LIN {X 0,Y 347.615,Z 494.435,A -85,B 0,C 180,E1 -13747.41,E2 -13747.41} C_VEL
LIN {X 0,Y 347.369,Z 499.212,A -85,B 0,C 180,E1 -13749.012,E2 -13749.012} C_VEL
LIN {X 0,Y 349.392,Z 514.132,A -85,B 0,C 180,E1 -13749.644,E2 -13749.644} C_VEL
LIN {X 0,Y 350.542,Z 527.666,A -85,B 0,C 180,E1 -13750.442,E2 -13750.442} C_VEL
LIN {X 0,Y 350.977,Z 539.209,A -85,B 0,C 180,E1 -13751.314,E2 -13751.314} C_VEL
LIN {X 0,Y 351.131,Z 550.524,A -85,B 0,C 180,E1 -13752.378,E2 -13752.378} C_VEL
LIN {X 0,Y 350.226,Z 559.587,A -85,B 0,C 180,E1 -13753.384,E2 -13753.384} C_VEL
LIN {X 0,Y 349.097,Z 570.237,A -85,B 0,C 180,E1 -13754.828,E2 -13754.828} C_VEL
LIN {X 0,Y 348.343,Z 577.267,A -85,B 0,C 180,E1 -13755.989,E2 -13755.989} C_VEL
LIN {X 0,Y 347.516,Z 586.102,A -85,B 0,C 180,E1 -13757.74,E2 -13757.74} C_VEL
LIN {X 0,Y 346.973,Z 593.197,A -85,B 0,C 180,E1 -13759.496,E2 -13759.496} C_VEL
LIN {X 0,Y 346.818,Z 598.935,A -85,B 0,C 180,E1 -13761.258,E2 -13761.258} C_VEL
LIN {X 0,Y 346.825,Z 603.831,A -85,B 0,C 180,E1 -13763.183,E2 -13763.183} C_VEL
LIN {X 0,Y 347.091,Z 607.836,A -85,B 0,C 180,E1 -13765.354,E2 -13765.354} C_VEL
LIN {X 0,Y 347.195,Z 609.309,A -85,B 0,C 180,E1 -13766.519,E2 -13766.519} C_VEL
LIN {X 0,Y 347.265,Z 610.359,A -85,B 0,C 180,E1 -13767.68,E2 -13767.68} C_VEL
LIN {X 0,Y 347.626,Z 611.268,A -85,B 0,C 180,E1 -13770,E2 -13770} C_VEL
LIN {X 0,Y 347.266,Z 610.353,A -85,B 0,C 180,E1 -13772.32,E2 -13772.32} C_VEL
LIN {X 0,Y 347.196,Z 609.302,A -85,B 0,C 180,E1 -13773.482,E2 -13773.482} C_VEL
LIN {X 0,Y 347.09,Z 607.824,A -85,B 0,C 180,E1 -13774.646,E2 -13774.646} C_VEL
LIN {X 0,Y 346.813,Z 603.843,A -85,B 0,C 180,E1 -13776.8,E2 -13776.8} C_VEL
LIN {X 0,Y 346.818,Z 598.902,A -85,B 0,C 180,E1 -13778.742,E2 -13778.742} C_VEL
LIN {X 0,Y 346.977,Z 593.158,A -85,B 0,C 180,E1 -13780.504,E2 -13780.504} C_VEL
LIN {X 0,Y 347.512,Z 586.051,A -85,B 0,C 180,E1 -13782.26,E2 -13782.26} C_VEL
LIN {X 0,Y 348.302,Z 577.193,A -85,B 0,C 180,E1 -13784.013,E2 -13784.013} C_VEL
LIN {X 0,Y 349.339,Z 568.176,A -85,B 0,C 180,E1 -13785.46,E2 -13785.46} C_VEL
LIN {X 0,Y 350.409,Z 558.302,A -85,B 0,C 180,E1 -13786.757,E2 -13786.757} C_VEL
LIN {X 0,Y 351.091,Z 550.396,A -85,B 0,C 180,E1 -13787.624,E2 -13787.624} C_VEL
LIN {X 0,Y 350.986,Z 539.051,A -85,B 0,C 180,E1 -13788.686,E2 -13788.686} C_VEL
LIN {X 0,Y 350.444,Z 525.95,A -85,B 0,C 180,E1 -13789.661,E2 -13789.661} C_VEL
LIN {X 0,Y 349.17,Z 512.232,A -85,B 0,C 180,E1 -13790.432,E2 -13790.432} C_VEL
LIN {X 0,Y 347.349,Z 499.21,A -85,B 0,C 180,E1 -13790.97,E2 -13790.97} C_VEL
LIN {X 0,Y 348.076,Z 488.085,A -85,B 0,C 180,E1 -13794.688,E2 -13794.688} C_VEL
LIN {X 0,Y 349.057,Z 475.439,A -85,B 0,C 180,E1 -13798.896,E2 -13798.896} C_VEL
LIN {X 0,Y 350.254,Z 463.775,A -85,B 0,C 180,E1 -13802.804,E2 -13802.804} C_VEL
LIN {X 0,Y 351.609,Z 451.807,A -85,B 0,C 180,E1 -13806.915,E2 -13806.915} C_VEL
LIN {X 0,Y 351.655,Z 448.004,A -85,B 0,C 180,E1 -13808.284,E2 -13808.284} C_VEL
LIN {X 0,Y 350.132,Z 439.763,A -85,B 0,C 180,E1 -13811.483,E2 -13811.483} C_VEL
LIN {X 0,Y 348.357,Z 431.103,A -85,B 0,C 180,E1 -13815.08,E2 -13815.08} C_VEL
LIN {X 0,Y 347.734,Z 428.173,A -85,B 0,C 180,E1 -13816.394,E2 -13816.394} C_VEL
LIN {X 0,Y 347.735,Z 428.172,A -85,B 0,C 180,E1 -13819.703,E2 -13819.703} C_VEL
LIN {X 0,Y 347.765,Z 428.164,A -85,B 0,C 180,E1 -13822.68,E2 -13822.68} C_VEL
LIN {X 0,Y 347.751,Z 428.17,A -85,B 0,C 180,E1 -13825.956,E2 -13825.956} C_VEL
LIN {X 0,Y 347.752,Z 428.167,A -85,B 0,C 180,E1 -13829.652,E2 -13829.652} C_VEL
LIN {X 0,Y 347.833,Z 428.157,A -85,B 0,C 180,E1 -13833.608,E2 -13833.608} C_VEL
LIN {X 0,Y 347.787,Z 428.164,A -85,B 0,C 180,E1 -13836.162,E2 -13836.162} C_VEL
LIN {X 0,Y 347.815,Z 428.162,A -85,B 0,C 180,E1 -13839.909,E2 -13839.909} C_VEL
LIN {X 0,Y 347.87,Z 428.151,A -85,B 0,C 180,E1 -13842.359,E2 -13842.359} C_VEL
LIN {X 0,Y 347.901,Z 428.15,A -85,B 0,C 180,E1 -13845.971,E2 -13845.971} C_VEL
LIN {X 0,Y 347.933,Z 428.146,A -85,B 0,C 180,E1 -13849.526,E2 -13849.526} C_VEL
LIN {X 0,Y 348.083,Z 428.124,A -85,B 0,C 180,E1 -13853.042,E2 -13853.042} C_VEL
LIN {X 0,Y 348.212,Z 428.113,A -85,B 0,C 180,E1 -13857.687,E2 -13857.687} C_VEL
LIN {X 0,Y 348.371,Z 428.089,A -85,B 0,C 180,E1 -13860,E2 -13860} C_VEL
LIN {X 0,Y 348.21,Z 428.108,A -85,B 0,C 180,E1 -13862.314,E2 -13862.314} C_VEL
LIN {X 0,Y 348.082,Z 428.124,A -85,B 0,C 180,E1 -13866.958,E2 -13866.958} C_VEL
LIN {X 0,Y 347.934,Z 428.141,A -85,B 0,C 180,E1 -13870.474,E2 -13870.474} C_VEL
LIN {X 0,Y 347.901,Z 428.143,A -85,B 0,C 180,E1 -13874.15,E2 -13874.15} C_VEL
LIN {X 0,Y 347.894,Z 428.145,A -85,B 0,C 180,E1 -13878.29,E2 -13878.29} C_VEL
LIN {X 0,Y 347.793,Z 428.162,A -85,B 0,C 180,E1 -13881.636,E2 -13881.636} C_VEL
LIN {X 0,Y 347.816,Z 428.159,A -85,B 0,C 180,E1 -13885.108,E2 -13885.108} C_VEL
LIN {X 0,Y 347.811,Z 428.156,A -85,B 0,C 180,E1 -13887.694,E2 -13887.694} C_VEL
LIN {X 0,Y 347.752,Z 428.163,A -85,B 0,C 180,E1 -13890.348,E2 -13890.348} C_VEL
LIN {X 0,Y 347.751,Z 428.164,A -85,B 0,C 180,E1 -13894.044,E2 -13894.044} C_VEL
LIN {X 0,Y 347.764,Z 428.167,A -85,B 0,C 180,E1 -13897.321,E2 -13897.321} C_VEL
LIN {X 0,Y 347.735,Z 428.166,A -85,B 0,C 180,E1 -13900.297,E2 -13900.297} C_VEL
LIN {X 0,Y 347.732,Z 428.169,A -85,B 0,C 180,E1 -13903.407,E2 -13903.407} C_VEL
LIN {X 0,Y 347.788,Z 428.162,A -85,B 0,C 180,E1 -13906.676,E2 -13906.676} C_VEL
LIN {X 0,Y 347.789,Z 428.159,A -85,B 0,C 180,E1 -13910.165,E2 -13910.165} C_VEL
LIN {X 0,Y 347.793,Z 428.159,A -85,B 0,C 180,E1 -13914.125,E2 -13914.125} C_VEL
LIN {X 0,Y 347.741,Z 428.165,A -85,B 0,C 180,E1 -13918.086,E2 -13918.086} C_VEL
LIN {X 0,Y 347.782,Z 428.166,A -85,B 0,C 180,E1 -13920.988,E2 -13920.988} C_VEL
LIN {X 0,Y 347.834,Z 428.155,A -85,B 0,C 180,E1 -13923.608,E2 -13923.608} C_VEL
LIN {X 0,Y 347.792,Z 428.16,A -85,B 0,C 180,E1 -13926.162,E2 -13926.162} C_VEL
LIN {X 0,Y 347.82,Z 428.157,A -85,B 0,C 180,E1 -13929.91,E2 -13929.91} C_VEL
LIN {X 0,Y 347.858,Z 428.349,A -85,B 0,C 180,E1 -13930.016,E2 -13930.016} C_VEL
LIN {X 0,Y 351.858,Z 440.054,A -85,B 0,C 180,E1 -13931.095,E2 -13931.095} C_VEL
LIN {X 0,Y 354.541,Z 449.162,A -85,B 0,C 180,E1 -13932.082,E2 -13932.082} C_VEL
LIN {X 0,Y 355.019,Z 451.116,A -85,B 0,C 180,E1 -13932.305,E2 -13932.305} C_VEL
LIN {X 0,Y 354.008,Z 461.436,A -85,B 0,C 180,E1 -13933.418,E2 -13933.418} C_VEL
LIN {X 0,Y 353.05,Z 471.021,A -85,B 0,C 180,E1 -13934.706,E2 -13934.706} C_VEL
LIN {X 0,Y 352.106,Z 479.723,A -85,B 0,C 180,E1 -13936.142,E2 -13936.142} C_VEL
LIN {X 0,Y 350.939,Z 488.223,A -85,B 0,C 180,E1 -13937.861,E2 -13937.861} C_VEL
LIN {X 0,Y 349.95,Z 495.551,A -85,B 0,C 180,E1 -13939.758,E2 -13939.758} C_VEL
LIN {X 0,Y 349.449,Z 500.347,A -85,B 0,C 180,E1 -13941.324,E2 -13941.324} C_VEL
LIN {X 0,Y 348.745,Z 504.594,A -85,B 0,C 180,E1 -13943.055,E2 -13943.055} C_VEL
LIN {X 0,Y 348.436,Z 506.829,A -85,B 0,C 180,E1 -13944.212,E2 -13944.212} C_VEL
LIN {X 0,Y 348.162,Z 508.651,A -85,B 0,C 180,E1 -13945.369,E2 -13945.369} C_VEL
LIN {X 0,Y 347.931,Z 510.025,A -85,B 0,C 180,E1 -13946.526,E2 -13946.526} C_VEL
LIN {X 0,Y 347.95,Z 511.562,A -85,B 0,C 180,E1 -13948.843,E2 -13948.843} C_VEL
LIN {X 0,Y 347.949,Z 511.785,A -85,B 0,C 180,E1 -13950,E2 -13950} C_VEL
LIN {X 0,Y 347.949,Z 511.603,A -85,B 0,C 180,E1 -13951.157,E2 -13951.157} C_VEL
LIN {X 0,Y 347.923,Z 510.12,A -85,B 0,C 180,E1 -13953.474,E2 -13953.474} C_VEL
LIN {X 0,Y 348.151,Z 508.789,A -85,B 0,C 180,E1 -13954.631,E2 -13954.631} C_VEL
LIN {X 0,Y 348.63,Z 505.972,A -85,B 0,C 180,E1 -13956.366,E2 -13956.366} C_VEL
LIN {X 0,Y 349.241,Z 502.154,A -85,B 0,C 180,E1 -13958.098,E2 -13958.098} C_VEL
LIN {X 0,Y 349.841,Z 496.248,A -85,B 0,C 180,E1 -13960.143,E2 -13960.143} C_VEL
LIN {X 0,Y 350.782,Z 489.852,A -85,B 0,C 180,E1 -13961.851,E2 -13961.851} C_VEL
LIN {X 0,Y 351.886,Z 481.818,A -85,B 0,C 180,E1 -13963.572,E2 -13963.572} C_VEL
LIN {X 0,Y 352.754,Z 473.601,A -85,B 0,C 180,E1 -13965.011,E2 -13965.011} C_VEL
LIN {X 0,Y 353.83,Z 463.41,A -85,B 0,C 180,E1 -13966.442,E2 -13966.442} C_VEL
LIN {X 0,Y 354.776,Z 453.903,A -85,B 0,C 180,E1 -13967.519,E2 -13967.519} C_VEL
LIN {X 0,Y 354.989,Z 450.779,A -85,B 0,C 180,E1 -13967.836,E2 -13967.836} C_VEL
LIN {X 0,Y 351.781,Z 439.815,A -85,B 0,C 180,E1 -13969.035,E2 -13969.035} C_VEL
LIN {X 0,Y 347.808,Z 428.164,A -85,B 0,C 180,E1 -13970.129,E2 -13970.129} C_VEL
LIN {X 0,Y 347.791,Z 428.161,A -85,B 0,C 180,E1 -13973.838,E2 -13973.838} C_VEL
LIN {X 0,Y 347.852,Z 428.157,A -85,B 0,C 180,E1 -13977.255,E2 -13977.255} C_VEL
LIN {X 0,Y 347.751,Z 428.164,A -85,B 0,C 180,E1 -13980.348,E2 -13980.348} C_VEL
LIN {X 0,Y 347.75,Z 428.164,A -85,B 0,C 180,E1 -13984.044,E2 -13984.044} C_VEL
LIN {X 0,Y 347.769,Z 428.166,A -85,B 0,C 180,E1 -13987.32,E2 -13987.32} C_VEL
LIN {X 0,Y 347.796,Z 428.159,A -85,B 0,C 180,E1 -13990.288,E2 -13990.288} C_VEL
LIN {X 0,Y 347.788,Z 428.162,A -85,B 0,C 180,E1 -13993.398,E2 -13993.398} C_VEL
LIN {X 0,Y 347.732,Z 428.17,A -85,B 0,C 180,E1 -13996.685,E2 -13996.685} C_VEL
LIN {X 0,Y 347.738,Z 428.166,A -85,B 0,C 180,E1 -13999.9,E2 -13999.9} C_VEL
LIN {X 0,Y 347.096,Z 428.251,A -85,B 0,C 180,E1 -14000.867,E2 -14000.867} C_VEL
LIN {X 0,Y 344.256,Z 428.605,A -85,B 0,C 180,E1 -14002.441,E2 -14002.441} C_VEL
LIN {X 0,Y 341.835,Z 428.908,A -85,B 0,C 180,E1 -14003.715,E2 -14003.715} C_VEL
LIN {X 0,Y 340.796,Z 429.035,A -85,B 0,C 180,E1 -14004.701,E2 -14004.701} C_VEL
LIN {X 0,Y 340.712,Z 429.043,A -85,B 0,C 180,E1 -14005.034,E2 -14005.034} C_VEL
LIN {X 0,Y 340.7,Z 429.048,A -85,B 0,C 180,E1 -14008.955,E2 -14008.955} C_VEL
LIN {X 0,Y 340.805,Z 429.033,A -85,B 0,C 180,E1 -14013.02,E2 -14013.02} C_VEL
LIN {X 0,Y 340.758,Z 429.035,A -85,B 0,C 180,E1 -14015.638,E2 -14015.638} C_VEL
LIN {X 0,Y 340.755,Z 429.036,A -85,B 0,C 180,E1 -14019.475,E2 -14019.475} C_VEL
LIN {X 0,Y 340.86,Z 429.023,A -85,B 0,C 180,E1 -14021.984,E2 -14021.984} C_VEL
LIN {X 0,Y 340.871,Z 429.021,A -85,B 0,C 180,E1 -14025.705,E2 -14025.705} C_VEL
LIN {X 0,Y 340.875,Z 429.021,A -85,B 0,C 180,E1 -14029.306,E2 -14029.306} C_VEL
LIN {X 0,Y 341.051,Z 429,A -85,B 0,C 180,E1 -14032.898,E2 -14032.898} C_VEL
LIN {X 0,Y 341.173,Z 428.984,A -85,B 0,C 180,E1 -14037.639,E2 -14037.639} C_VEL
LIN {X 0,Y 341.319,Z 428.968,A -85,B 0,C 180,E1 -14040,E2 -14040} C_VEL
LIN {X 0,Y 341.173,Z 428.988,A -85,B 0,C 180,E1 -14042.361,E2 -14042.361} C_VEL
LIN {X 0,Y 341.049,Z 428.999,A -85,B 0,C 180,E1 -14047.102,E2 -14047.102} C_VEL
LIN {X 0,Y 340.875,Z 429.023,A -85,B 0,C 180,E1 -14050.694,E2 -14050.694} C_VEL
LIN {X 0,Y 340.865,Z 429.027,A -85,B 0,C 180,E1 -14054.325,E2 -14054.325} C_VEL
LIN {X 0,Y 340.84,Z 429.029,A -85,B 0,C 180,E1 -14058.467,E2 -14058.467} C_VEL
LIN {X 0,Y 340.719,Z 429.044,A -85,B 0,C 180,E1 -14061.842,E2 -14061.842} C_VEL
LIN {X 0,Y 340.773,Z 429.036,A -85,B 0,C 180,E1 -14065.664,E2 -14065.664} C_VEL
LIN {X 0,Y 340.731,Z 429.042,A -85,B 0,C 180,E1 -14068.321,E2 -14068.321} C_VEL
LIN {X 0,Y 340.699,Z 429.043,A -85,B 0,C 180,E1 -14071.045,E2 -14071.045} C_VEL
LIN {X 0,Y 340.72,Z 429.042,A -85,B 0,C 180,E1 -14075.279,E2 -14075.279} C_VEL
LIN {X 0,Y 340.712,Z 429.044,A -85,B 0,C 180,E1 -14078.386,E2 -14078.386} C_VEL
LIN {X 0,Y 340.701,Z 429.05,A -85,B 0,C 180,E1 -14082.046,E2 -14082.046} C_VEL
LIN {X 0,Y 340.693,Z 429.067,A -85,B 0,C 180,E1 -14083.145,E2 -14083.145} C_VEL
LIN {X 0,Y 342.387,Z 437.143,A -85,B 0,C 180,E1 -14086.699,E2 -14086.699} C_VEL
LIN {X 0,Y 343.982,Z 445.1,A -85,B 0,C 180,E1 -14089.972,E2 -14089.972} C_VEL
LIN {X 0,Y 344.84,Z 451.146,A -85,B 0,C 180,E1 -14092.308,E2 -14092.308} C_VEL
LIN {X 0,Y 343.637,Z 460.942,A -85,B 0,C 180,E1 -14095.776,E2 -14095.776} C_VEL
LIN {X 0,Y 342.775,Z 468.732,A -85,B 0,C 180,E1 -14098.478,E2 -14098.478} C_VEL
LIN {X 0,Y 341.626,Z 480.835,A -85,B 0,C 180,E1 -14102.627,E2 -14102.627} C_VEL
LIN {X 0,Y 340.803,Z 491.561,A -85,B 0,C 180,E1 -14106.289,E2 -14106.289} C_VEL
LIN {X 0,Y 340.351,Z 498.191,A -85,B 0,C 180,E1 -14108.568,E2 -14108.568} C_VEL
LIN {X 0,Y 342.379,Z 512.492,A -85,B 0,C 180,E1 -14109.184,E2 -14109.184} C_VEL
LIN {X 0,Y 343.496,Z 525.586,A -85,B 0,C 180,E1 -14109.955,E2 -14109.955} C_VEL
LIN {X 0,Y 344.073,Z 538.171,A -85,B 0,C 180,E1 -14110.924,E2 -14110.924} C_VEL
LIN {X 0,Y 344.161,Z 550.943,A -85,B 0,C 180,E1 -14112.163,E2 -14112.163} C_VEL
LIN {X 0,Y 343.238,Z 559.759,A -85,B 0,C 180,E1 -14113.189,E2 -14113.189} C_VEL
LIN {X 0,Y 342.06,Z 570.288,A -85,B 0,C 180,E1 -14114.686,E2 -14114.686} C_VEL
LIN {X 0,Y 341.269,Z 577.873,A -85,B 0,C 180,E1 -14115.997,E2 -14115.997} C_VEL
LIN {X 0,Y 340.406,Z 586.348,A -85,B 0,C 180,E1 -14117.783,E2 -14117.783} C_VEL
LIN {X 0,Y 339.886,Z 593.222,A -85,B 0,C 180,E1 -14119.576,E2 -14119.576} C_VEL
LIN {X 0,Y 339.731,Z 599.572,A -85,B 0,C 180,E1 -14121.674,E2 -14121.674} C_VEL
LIN {X 0,Y 339.756,Z 603.095,A -85,B 0,C 180,E1 -14123.17,E2 -14123.17} C_VEL
LIN {X 0,Y 340.028,Z 606.823,A -85,B 0,C 180,E1 -14125.258,E2 -14125.258} C_VEL
LIN {X 0,Y 340.147,Z 608.299,A -85,B 0,C 180,E1 -14126.446,E2 -14126.446} C_VEL
LIN {X 0,Y 340.221,Z 609.351,A -85,B 0,C 180,E1 -14127.632,E2 -14127.632} C_VEL
LIN {X 0,Y 340.597,Z 610.263,A -85,B 0,C 180,E1 -14130,E2 -14130} C_VEL
LIN {X 0,Y 340.222,Z 609.345,A -85,B 0,C 180,E1 -14132.368,E2 -14132.368} C_VEL
LIN {X 0,Y 340.147,Z 608.291,A -85,B 0,C 180,E1 -14133.554,E2 -14133.554} C_VEL
LIN {X 0,Y 340.027,Z 606.81,A -85,B 0,C 180,E1 -14134.743,E2 -14134.743} C_VEL
LIN {X 0,Y 339.75,Z 603.089,A -85,B 0,C 180,E1 -14136.821,E2 -14136.821} C_VEL
LIN {X 0,Y 339.742,Z 597.877,A -85,B 0,C 180,E1 -14138.925,E2 -14138.925} C_VEL
LIN {X 0,Y 339.937,Z 592.133,A -85,B 0,C 180,E1 -14140.724,E2 -14140.724} C_VEL
LIN {X 0,Y 340.505,Z 585.023,A -85,B 0,C 180,E1 -14142.517,E2 -14142.517} C_VEL
LIN {X 0,Y 341.232,Z 577.802,A -85,B 0,C 180,E1 -14144.005,E2 -14144.005} C_VEL
LIN {X 0,Y 342.036,Z 570.341,A -85,B 0,C 180,E1 -14145.293,E2 -14145.293} C_VEL
LIN {X 0,Y 343.041,Z 560.804,A -85,B 0,C 180,E1 -14146.668,E2 -14146.668} C_VEL
LIN {X 0,Y 344.134,Z 550.811,A -85,B 0,C 180,E1 -14147.839,E2 -14147.839} C_VEL
LIN {X 0,Y 344.045,Z 537.997,A -85,B 0,C 180,E1 -14149.077,E2 -14149.077} C_VEL
LIN {X 0,Y 343.509,Z 525.338,A -85,B 0,C 180,E1 -14150.045,E2 -14150.045} C_VEL
LIN {X 0,Y 342.262,Z 511.646,A -85,B 0,C 180,E1 -14150.843,E2 -14150.843} C_VEL
LIN {X 0,Y 340.324,Z 498.16,A -85,B 0,C 180,E1 -14151.422,E2 -14151.422} C_VEL
LIN {X 0,Y 341.221,Z 485.908,A -85,B 0,C 180,E1 -14155.628,E2 -14155.628} C_VEL
LIN {X 0,Y 342.144,Z 474.463,A -85,B 0,C 180,E1 -14159.537,E2 -14159.537} C_VEL
LIN {X 0,Y 343.266,Z 464.612,A -85,B 0,C 180,E1 -14162.92,E2 -14162.92} C_VEL
LIN {X 0,Y 344.722,Z 452.086,A -85,B 0,C 180,E1 -14167.334,E2 -14167.334} C_VEL
LIN {X 0,Y 344.678,Z 449.176,A -85,B 0,C 180,E1 -14168.408,E2 -14168.408} C_VEL
LIN {X 0,Y 343.159,Z 440.988,A -85,B 0,C 180,E1 -14171.664,E2 -14171.664} C_VEL
LIN {X 0,Y 341.562,Z 433.244,A -85,B 0,C 180,E1 -14174.955,E2 -14174.955} C_VEL
LIN {X 0,Y 340.674,Z 429.052,A -85,B 0,C 180,E1 -14176.854,E2 -14176.854} C_VEL
LIN {X 0,Y 340.702,Z 429.049,A -85,B 0,C 180,E1 -14180.248,E2 -14180.248} C_VEL
LIN {X 0,Y 340.713,Z 429.043,A -85,B 0,C 180,E1 -14183.559,E2 -14183.559} C_VEL
LIN {X 0,Y 340.697,Z 429.048,A -85,B 0,C 180,E1 -14186.154,E2 -14186.154} C_VEL
LIN {X 0,Y 340.744,Z 429.041,A -85,B 0,C 180,E1 -14190.329,E2 -14190.329} C_VEL
LIN {X 0,Y 340.806,Z 429.03,A -85,B 0,C 180,E1 -14193.02,E2 -14193.02} C_VEL
LIN {X 0,Y 340.757,Z 429.039,A -85,B 0,C 180,E1 -14195.638,E2 -14195.638} C_VEL
LIN {X 0,Y 340.74,Z 429.04,A -85,B 0,C 180,E1 -14199.474,E2 -14199.474} C_VEL
LIN {X 0,Y 340.861,Z 429.028,A -85,B 0,C 180,E1 -14201.984,E2 -14201.984} C_VEL
LIN {X 0,Y 340.872,Z 429.027,A -85,B 0,C 180,E1 -14205.705,E2 -14205.705} C_VEL
LIN {X 0,Y 340.876,Z 429.023,A -85,B 0,C 180,E1 -14209.306,E2 -14209.306} C_VEL
LIN {X 0,Y 341.05,Z 429,A -85,B 0,C 180,E1 -14212.898,E2 -14212.898} C_VEL
LIN {X 0,Y 341.174,Z 428.989,A -85,B 0,C 180,E1 -14217.639,E2 -14217.639} C_VEL
LIN {X 0,Y 341.32,Z 428.968,A -85,B 0,C 180,E1 -14220,E2 -14220} C_VEL
LIN {X 0,Y 341.172,Z 428.984,A -85,B 0,C 180,E1 -14222.361,E2 -14222.361} C_VEL
LIN {X 0,Y 341.05,Z 429.001,A -85,B 0,C 180,E1 -14227.102,E2 -14227.102} C_VEL
LIN {X 0,Y 340.877,Z 429.021,A -85,B 0,C 180,E1 -14230.694,E2 -14230.694} C_VEL
LIN {X 0,Y 340.866,Z 429.018,A -85,B 0,C 180,E1 -14234.325,E2 -14234.325} C_VEL
LIN {X 0,Y 340.84,Z 429.023,A -85,B 0,C 180,E1 -14238.466,E2 -14238.466} C_VEL
LIN {X 0,Y 340.757,Z 429.037,A -85,B 0,C 180,E1 -14241.857,E2 -14241.857} C_VEL
LIN {X 0,Y 340.776,Z 429.033,A -85,B 0,C 180,E1 -14245.664,E2 -14245.664} C_VEL
LIN {X 0,Y 340.731,Z 429.034,A -85,B 0,C 180,E1 -14248.321,E2 -14248.321} C_VEL
LIN {X 0,Y 340.701,Z 429.045,A -85,B 0,C 180,E1 -14251.045,E2 -14251.045} C_VEL
LIN {X 0,Y 340.721,Z 429.045,A -85,B 0,C 180,E1 -14255.279,E2 -14255.279} C_VEL
LIN {X 0,Y 340.712,Z 429.042,A -85,B 0,C 180,E1 -14258.386,E2 -14258.386} C_VEL
LIN {X 0,Y 340.702,Z 429.042,A -85,B 0,C 180,E1 -14262.046,E2 -14262.046} C_VEL
LIN {X 0,Y 340.724,Z 429.042,A -85,B 0,C 180,E1 -14265.468,E2 -14265.468} C_VEL
LIN {X 0,Y 340.728,Z 429.042,A -85,B 0,C 180,E1 -14268.696,E2 -14268.696} C_VEL
LIN {X 0,Y 340.744,Z 429.037,A -85,B 0,C 180,E1 -14271.774,E2 -14271.774} C_VEL
LIN {X 0,Y 340.726,Z 429.039,A -85,B 0,C 180,E1 -14275.595,E2 -14275.595} C_VEL
LIN {X 0,Y 340.7,Z 429.048,A -85,B 0,C 180,E1 -14278.955,E2 -14278.955} C_VEL
LIN {X 0,Y 340.806,Z 429.035,A -85,B 0,C 180,E1 -14283.02,E2 -14283.02} C_VEL
LIN {X 0,Y 340.759,Z 429.036,A -85,B 0,C 180,E1 -14285.638,E2 -14285.638} C_VEL
LIN {X 0,Y 340.763,Z 429.036,A -85,B 0,C 180,E1 -14289.543,E2 -14289.543} C_VEL
LIN {X 0,Y 344.712,Z 440.423,A -85,B 0,C 180,E1 -14290.631,E2 -14290.631} C_VEL
LIN {X 0,Y 347.762,Z 450.74,A -85,B 0,C 180,E1 -14291.776,E2 -14291.776} C_VEL
LIN {X 0,Y 348.214,Z 452.481,A -85,B 0,C 180,E1 -14291.983,E2 -14291.983} C_VEL
LIN {X 0,Y 347.178,Z 463.595,A -85,B 0,C 180,E1 -14293.234,E2 -14293.234} C_VEL
LIN {X 0,Y 346.063,Z 473.943,A -85,B 0,C 180,E1 -14294.692,E2 -14294.692} C_VEL
LIN {X 0,Y 345.095,Z 482.305,A -85,B 0,C 180,E1 -14296.155,E2 -14296.155} C_VEL
LIN {X 0,Y 343.912,Z 490.435,A -85,B 0,C 180,E1 -14297.909,E2 -14297.909} C_VEL
LIN {X 0,Y 343.036,Z 496.558,A -85,B 0,C 180,E1 -14299.55,E2 -14299.55} C_VEL
LIN {X 0,Y 342.504,Z 501.354,A -85,B 0,C 180,E1 -14301.147,E2 -14301.147} C_VEL
LIN {X 0,Y 341.772,Z 505.6,A -85,B 0,C 180,E1 -14302.913,E2 -14302.913} C_VEL
LIN {X 0,Y 341.445,Z 507.835,A -85,B 0,C 180,E1 -14304.093,E2 -14304.093} C_VEL
LIN {X 0,Y 341.157,Z 509.657,A -85,B 0,C 180,E1 -14305.273,E2 -14305.273} C_VEL
LIN {X 0,Y 340.916,Z 511.031,A -85,B 0,C 180,E1 -14306.454,E2 -14306.454} C_VEL
LIN {X 0,Y 340.931,Z 512.566,A -85,B 0,C 180,E1 -14308.819,E2 -14308.819} C_VEL
LIN {X 0,Y 340.928,Z 512.79,A -85,B 0,C 180,E1 -14310,E2 -14310} C_VEL
LIN {X 0,Y 340.931,Z 512.607,A -85,B 0,C 180,E1 -14311.181,E2 -14311.181} C_VEL
LIN {X 0,Y 340.909,Z 511.125,A -85,B 0,C 180,E1 -14313.546,E2 -14313.546} C_VEL
LIN {X 0,Y 341.146,Z 509.793,A -85,B 0,C 180,E1 -14314.727,E2 -14314.727} C_VEL
LIN {X 0,Y 341.648,Z 506.976,A -85,B 0,C 180,E1 -14316.496,E2 -14316.496} C_VEL
LIN {X 0,Y 342.284,Z 503.158,A -85,B 0,C 180,E1 -14318.264,E2 -14318.264} C_VEL
LIN {X 0,Y 342.924,Z 497.255,A -85,B 0,C 180,E1 -14320.349,E2 -14320.349} C_VEL
LIN {X 0,Y 343.907,Z 490.855,A -85,B 0,C 180,E1 -14322.091,E2 -14322.091} C_VEL
LIN {X 0,Y 345.058,Z 482.82,A -85,B 0,C 180,E1 -14323.846,E2 -14323.846} C_VEL
LIN {X 0,Y 345.971,Z 474.603,A -85,B 0,C 180,E1 -14325.312,E2 -14325.312} C_VEL
LIN {X 0,Y 347.095,Z 464.411,A -85,B 0,C 180,E1 -14326.77,E2 -14326.77} C_VEL
LIN {X 0,Y 348.141,Z 454.319,A -85,B 0,C 180,E1 -14327.927,E2 -14327.927} C_VEL
LIN {X 0,Y 348.212,Z 452.186,A -85,B 0,C 180,E1 -14328.155,E2 -14328.155} C_VEL
LIN {X 0,Y 344.956,Z 441.235,A -85,B 0,C 180,E1 -14329.396,E2 -14329.396} C_VEL
LIN {X 0,Y 340.788,Z 429.038,A -85,B 0,C 180,E1 -14330.563,E2 -14330.563} C_VEL
LIN {X 0,Y 340.769,Z 429.037,A -85,B 0,C 180,E1 -14334.844,E2 -14334.844} C_VEL
LIN {X 0,Y 340.778,Z 429.035,A -85,B 0,C 180,E1 -14337.525,E2 -14337.525} C_VEL
LIN {X 0,Y 340.7,Z 429.047,A -85,B 0,C 180,E1 -14341.044,E2 -14341.044} C_VEL
LIN {X 0,Y 340.721,Z 429.045,A -85,B 0,C 180,E1 -14345.279,E2 -14345.279} C_VEL
LIN {X 0,Y 340.727,Z 429.04,A -85,B 0,C 180,E1 -14348.389,E2 -14348.389} C_VEL
LIN {X 0,Y 340.728,Z 429.043,A -85,B 0,C 180,E1 -14351.303,E2 -14351.303} C_VEL
LIN {X 0,Y 340.724,Z 429.041,A -85,B 0,C 180,E1 -14354.532,E2 -14354.532} C_VEL
LIN {X 0,Y 340.688,Z 429.047,A -85,B 0,C 180,E1 -14358.691,E2 -14358.691} C_VEL
LIN {X 0,Y 340.735,Z 429.039,A -85,B 0,C 180,E1 -14361.773,E2 -14361.773} C_VEL
LIN {X 0,Y 340.712,Z 429.043,A -85,B 0,C 180,E1 -14365.034,E2 -14365.034} C_VEL
LIN {X 0,Y 340.049,Z 429.125,A -85,B 0,C 180,E1 -14366.021,E2 -14366.021} C_VEL
LIN {X 0,Y 337.206,Z 429.477,A -85,B 0,C 180,E1 -14367.626,E2 -14367.626} C_VEL
LIN {X 0,Y 334.794,Z 429.784,A -85,B 0,C 180,E1 -14368.925,E2 -14368.925} C_VEL
LIN {X 0,Y 333.758,Z 429.908,A -85,B 0,C 180,E1 -14369.931,E2 -14369.931} C_VEL
LIN {X 0,Y 333.673,Z 429.917,A -85,B 0,C 180,E1 -14370.271,E2 -14370.271} C_VEL
LIN {X 0,Y 333.737,Z 429.91,A -85,B 0,C 180,E1 -14373.754,E2 -14373.754} C_VEL
LIN {X 0,Y 333.721,Z 429.911,A -85,B 0,C 180,E1 -14377.914,E2 -14377.914} C_VEL
LIN {X 0,Y 333.796,Z 429.902,A -85,B 0,C 180,E1 -14381.589,E2 -14381.589} C_VEL
LIN {X 0,Y 333.81,Z 429.901,A -85,B 0,C 180,E1 -14385.576,E2 -14385.576} C_VEL
LIN {X 0,Y 333.838,Z 429.898,A -85,B 0,C 180,E1 -14389.078,E2 -14389.078} C_VEL
LIN {X 0,Y 333.997,Z 429.88,A -85,B 0,C 180,E1 -14392.747,E2 -14392.747} C_VEL
LIN {X 0,Y 333.811,Z 429.899,A -85,B 0,C 180,E1 -14395.169,E2 -14395.169} C_VEL
LIN {X 0,Y 334.11,Z 429.864,A -85,B 0,C 180,E1 -14397.589,E2 -14397.589} C_VEL
LIN {X 0,Y 334.269,Z 429.846,A -85,B 0,C 180,E1 -14400,E2 -14400} C_VEL
LIN {X 0,Y 334.11,Z 429.868,A -85,B 0,C 180,E1 -14402.411,E2 -14402.411} C_VEL
LIN {X 0,Y 334.012,Z 429.879,A -85,B 0,C 180,E1 -14406.039,E2 -14406.039} C_VEL
LIN {X 0,Y 333.852,Z 429.897,A -85,B 0,C 180,E1 -14409.695,E2 -14409.695} C_VEL
LIN {X 0,Y 333.801,Z 429.902,A -85,B 0,C 180,E1 -14413.391,E2 -14413.391} C_VEL
LIN {X 0,Y 333.749,Z 429.908,A -85,B 0,C 180,E1 -14417.146,E2 -14417.146} C_VEL
LIN {X 0,Y 333.737,Z 429.912,A -85,B 0,C 180,E1 -14419.69,E2 -14419.69} C_VEL
LIN {X 0,Y 333.671,Z 429.92,A -85,B 0,C 180,E1 -14423.59,E2 -14423.59} C_VEL
LIN {X 0,Y 333.737,Z 429.915,A -85,B 0,C 180,E1 -14426.246,E2 -14426.246} C_VEL
LIN {X 0,Y 333.692,Z 429.916,A -85,B 0,C 180,E1 -14428.974,E2 -14428.974} C_VEL
LIN {X 0,Y 333.647,Z 429.923,A -85,B 0,C 180,E1 -14432.588,E2 -14432.588} C_VEL
LIN {X 0,Y 333.678,Z 429.922,A -85,B 0,C 180,E1 -14436.139,E2 -14436.139} C_VEL
LIN {X 0,Y 333.648,Z 429.923,A -85,B 0,C 180,E1 -14439.192,E2 -14439.192} C_VEL
LIN {X 0,Y 333.671,Z 430.02,A -85,B 0,C 180,E1 -14442.701,E2 -14442.701} C_VEL
LIN {X 0,Y 335.277,Z 437.819,A -85,B 0,C 180,E1 -14446.232,E2 -14446.232} C_VEL
LIN {X 0,Y 336.937,Z 446.061,A -85,B 0,C 180,E1 -14449.713,E2 -14449.713} C_VEL
LIN {X 0,Y 337.881,Z 452.381,A -85,B 0,C 180,E1 -14452.224,E2 -14452.224} C_VEL
LIN {X 0,Y 336.432,Z 463.536,A -85,B 0,C 180,E1 -14456.255,E2 -14456.255} C_VEL
LIN {X 0,Y 335.296,Z 473.537,A -85,B 0,C 180,E1 -14459.798,E2 -14459.798} C_VEL
LIN {X 0,Y 334.265,Z 484.934,A -85,B 0,C 180,E1 -14463.798,E2 -14463.798} C_VEL
LIN {X 0,Y 333.399,Z 496.035,A -85,B 0,C 180,E1 -14467.701,E2 -14467.701} C_VEL
LIN {X 0,Y 333.318,Z 497.121,A -85,B 0,C 180,E1 -14468.086,E2 -14468.086} C_VEL
LIN {X 0,Y 335.461,Z 512.026,A -85,B 0,C 180,E1 -14468.759,E2 -14468.759} C_VEL
LIN {X 0,Y 336.521,Z 523.731,A -85,B 0,C 180,E1 -14469.468,E2 -14469.468} C_VEL
LIN {X 0,Y 337.141,Z 535.894,A -85,B 0,C 180,E1 -14470.409,E2 -14470.409} C_VEL
LIN {X 0,Y 337.147,Z 548.43,A -85,B 0,C 180,E1 -14471.622,E2 -14471.622} C_VEL
LIN {X 0,Y 337.019,Z 553.89,A -85,B 0,C 180,E1 -14472.243,E2 -14472.243} C_VEL
LIN {X 0,Y 335.774,Z 564.224,A -85,B 0,C 180,E1 -14473.587,E2 -14473.587} C_VEL
LIN {X 0,Y 334.6,Z 573.384,A -85,B 0,C 180,E1 -14475.059,E2 -14475.059} C_VEL
LIN {X 0,Y 333.796,Z 581.305,A -85,B 0,C 180,E1 -14476.609,E2 -14476.609} C_VEL
LIN {X 0,Y 333.081,Z 588.943,A -85,B 0,C 180,E1 -14478.437,E2 -14478.437} C_VEL
LIN {X 0,Y 332.729,Z 595.125,A -85,B 0,C 180,E1 -14480.272,E2 -14480.272} C_VEL
LIN {X 0,Y 332.669,Z 600.048,A -85,B 0,C 180,E1 -14482.107,E2 -14482.107} C_VEL
LIN {X 0,Y 332.767,Z 603.835,A -85,B 0,C 180,E1 -14483.938,E2 -14483.938} C_VEL
LIN {X 0,Y 332.966,Z 605.81,A -85,B 0,C 180,E1 -14485.157,E2 -14485.157} C_VEL
LIN {X 0,Y 333.098,Z 607.29,A -85,B 0,C 180,E1 -14486.371,E2 -14486.371} C_VEL
LIN {X 0,Y 333.176,Z 608.343,A -85,B 0,C 180,E1 -14487.582,E2 -14487.582} C_VEL
LIN {X 0,Y 333.568,Z 609.257,A -85,B 0,C 180,E1 -14490,E2 -14490} C_VEL
LIN {X 0,Y 333.177,Z 608.336,A -85,B 0,C 180,E1 -14492.418,E2 -14492.418} C_VEL
LIN {X 0,Y 333.098,Z 607.281,A -85,B 0,C 180,E1 -14493.629,E2 -14493.629} C_VEL
LIN {X 0,Y 332.966,Z 605.796,A -85,B 0,C 180,E1 -14494.843,E2 -14494.843} C_VEL
LIN {X 0,Y 332.682,Z 602.349,A -85,B 0,C 180,E1 -14496.836,E2 -14496.836} C_VEL
LIN {X 0,Y 332.663,Z 598.518,A -85,B 0,C 180,E1 -14498.505,E2 -14498.505} C_VEL
LIN {X 0,Y 332.857,Z 592.155,A -85,B 0,C 180,E1 -14500.647,E2 -14500.647} C_VEL
LIN {X 0,Y 333.394,Z 585.267,A -85,B 0,C 180,E1 -14502.479,E2 -14502.479} C_VEL
LIN {X 0,Y 334.149,Z 578.303,A -85,B 0,C 180,E1 -14503.997,E2 -14503.997} C_VEL
LIN {X 0,Y 334.511,Z 573.631,A -85,B 0,C 180,E1 -14504.883,E2 -14504.883} C_VEL
LIN {X 0,Y 335.772,Z 564.126,A -85,B 0,C 180,E1 -14506.414,E2 -14506.414} C_VEL
LIN {X 0,Y 336.991,Z 553.759,A -85,B 0,C 180,E1 -14507.759,E2 -14507.759} C_VEL
LIN {X 0,Y 337.15,Z 542.134,A -85,B 0,C 180,E1 -14509.009,E2 -14509.009} C_VEL
LIN {X 0,Y 336.894,Z 529.996,A -85,B 0,C 180,E1 -14510.059,E2 -14510.059} C_VEL
LIN {X 0,Y 335.93,Z 516.65,A -85,B 0,C 180,E1 -14510.962,E2 -14510.962} C_VEL
LIN {X 0,Y 334.221,Z 503.192,A -85,B 0,C 180,E1 -14511.652,E2 -14511.652} C_VEL
LIN {X 0,Y 333.304,Z 497.08,A -85,B 0,C 180,E1 -14511.909,E2 -14511.909} C_VEL
LIN {X 0,Y 334.141,Z 486.457,A -85,B 0,C 180,E1 -14515.647,E2 -14515.647} C_VEL
LIN {X 0,Y 335.077,Z 475.372,A -85,B 0,C 180,E1 -14519.531,E2 -14519.531} C_VEL
LIN {X 0,Y 336.306,Z 464.717,A -85,B 0,C 180,E1 -14523.29,E2 -14523.29} C_VEL
LIN {X 0,Y 337.642,Z 454.079,A -85,B 0,C 180,E1 -14527.131,E2 -14527.131} C_VEL
LIN {X 0,Y 337.796,Z 451.401,A -85,B 0,C 180,E1 -14528.131,E2 -14528.131} C_VEL
LIN {X 0,Y 336.707,Z 444.824,A -85,B 0,C 180,E1 -14530.769,E2 -14530.769} C_VEL
LIN {X 0,Y 334.925,Z 436.128,A -85,B 0,C 180,E1 -14534.484,E2 -14534.484} C_VEL
LIN {X 0,Y 333.646,Z 429.926,A -85,B 0,C 180,E1 -14537.397,E2 -14537.397} C_VEL
LIN {X 0,Y 333.655,Z 429.923,A -85,B 0,C 180,E1 -14541.202,E2 -14541.202} C_VEL
LIN {X 0,Y 333.679,Z 429.922,A -85,B 0,C 180,E1 -14543.861,E2 -14543.861} C_VEL
LIN {X 0,Y 333.648,Z 429.922,A -85,B 0,C 180,E1 -14547.412,E2 -14547.412} C_VEL
LIN {X 0,Y 333.692,Z 429.917,A -85,B 0,C 180,E1 -14551.026,E2 -14551.026} C_VEL
LIN {X 0,Y 333.737,Z 429.915,A -85,B 0,C 180,E1 -14553.754,E2 -14553.754} C_VEL
LIN {X 0,Y 333.659,Z 429.924,A -85,B 0,C 180,E1 -14557.719,E2 -14557.719} C_VEL
LIN {X 0,Y 333.798,Z 429.906,A -85,B 0,C 180,E1 -14561.59,E2 -14561.59} C_VEL
LIN {X 0,Y 333.811,Z 429.905,A -85,B 0,C 180,E1 -14565.577,E2 -14565.577} C_VEL
LIN {X 0,Y 333.839,Z 429.899,A -85,B 0,C 180,E1 -14569.078,E2 -14569.078} C_VEL
LIN {X 0,Y 333.997,Z 429.878,A -85,B 0,C 180,E1 -14572.747,E2 -14572.747} C_VEL
LIN {X 0,Y 333.814,Z 429.902,A -85,B 0,C 180,E1 -14575.169,E2 -14575.169} C_VEL
LIN {X 0,Y 334.111,Z 429.869,A -85,B 0,C 180,E1 -14577.589,E2 -14577.589} C_VEL
LIN {X 0,Y 334.27,Z 429.846,A -85,B 0,C 180,E1 -14580,E2 -14580} C_VEL
LIN {X 0,Y 334.109,Z 429.864,A -85,B 0,C 180,E1 -14582.411,E2 -14582.411} C_VEL
LIN {X 0,Y 333.986,Z 429.879,A -85,B 0,C 180,E1 -14586.627,E2 -14586.627} C_VEL
LIN {X 0,Y 333.853,Z 429.899,A -85,B 0,C 180,E1 -14589.695,E2 -14589.695} C_VEL
LIN {X 0,Y 333.802,Z 429.903,A -85,B 0,C 180,E1 -14593.391,E2 -14593.391} C_VEL
LIN {X 0,Y 333.75,Z 429.905,A -85,B 0,C 180,E1 -14597.146,E2 -14597.146} C_VEL
LIN {X 0,Y 333.742,Z 429.911,A -85,B 0,C 180,E1 -14599.69,E2 -14599.69} C_VEL
LIN {X 0,Y 333.696,Z 429.915,A -85,B 0,C 180,E1 -14602.278,E2 -14602.278} C_VEL
LIN {X 0,Y 333.738,Z 429.906,A -85,B 0,C 180,E1 -14606.246,E2 -14606.246} C_VEL
LIN {X 0,Y 333.693,Z 429.913,A -85,B 0,C 180,E1 -14608.974,E2 -14608.974} C_VEL
LIN {X 0,Y 333.646,Z 429.922,A -85,B 0,C 180,E1 -14612.587,E2 -14612.587} C_VEL
LIN {X 0,Y 333.679,Z 429.917,A -85,B 0,C 180,E1 -14616.139,E2 -14616.139} C_VEL
LIN {X 0,Y 333.649,Z 429.926,A -85,B 0,C 180,E1 -14619.192,E2 -14619.192} C_VEL
LIN {X 0,Y 333.637,Z 429.924,A -85,B 0,C 180,E1 -14622.5,E2 -14622.5} C_VEL
LIN {X 0,Y 333.672,Z 429.918,A -85,B 0,C 180,E1 -14625.967,E2 -14625.967} C_VEL
LIN {X 0,Y 333.704,Z 429.916,A -85,B 0,C 180,E1 -14629.304,E2 -14629.304} C_VEL
LIN {X 0,Y 333.67,Z 429.921,A -85,B 0,C 180,E1 -14633.167,E2 -14633.167} C_VEL
LIN {X 0,Y 333.639,Z 429.926,A -85,B 0,C 180,E1 -14636.792,E2 -14636.792} C_VEL
LIN {X 0,Y 333.697,Z 429.915,A -85,B 0,C 180,E1 -14639.713,E2 -14639.713} C_VEL
LIN {X 0,Y 333.742,Z 429.912,A -85,B 0,C 180,E1 -14642.401,E2 -14642.401} C_VEL
LIN {X 0,Y 333.73,Z 429.914,A -85,B 0,C 180,E1 -14645.091,E2 -14645.091} C_VEL
LIN {X 0,Y 333.699,Z 429.968,A -85,B 0,C 180,E1 -14649.094,E2 -14649.094} C_VEL
LIN {X 0,Y 337.883,Z 441.861,A -85,B 0,C 180,E1 -14650.255,E2 -14650.255} C_VEL
LIN {X 0,Y 341.01,Z 452.223,A -85,B 0,C 180,E1 -14651.448,E2 -14651.448} C_VEL
LIN {X 0,Y 341.409,Z 453.943,A -85,B 0,C 180,E1 -14651.66,E2 -14651.66} C_VEL
LIN {X 0,Y 340.455,Z 464.604,A -85,B 0,C 180,E1 -14652.893,E2 -14652.893} C_VEL
LIN {X 0,Y 339.292,Z 474.951,A -85,B 0,C 180,E1 -14654.378,E2 -14654.378} C_VEL
LIN {X 0,Y 338.279,Z 483.312,A -85,B 0,C 180,E1 -14655.87,E2 -14655.87} C_VEL
LIN {X 0,Y 337.044,Z 491.442,A -85,B 0,C 180,E1 -14657.659,E2 -14657.659} C_VEL
LIN {X 0,Y 336.127,Z 497.565,A -85,B 0,C 180,E1 -14659.332,E2 -14659.332} C_VEL
LIN {X 0,Y 335.561,Z 502.36,A -85,B 0,C 180,E1 -14660.962,E2 -14660.962} C_VEL
LIN {X 0,Y 334.801,Z 506.606,A -85,B 0,C 180,E1 -14662.764,E2 -14662.764} C_VEL
LIN {X 0,Y 334.455,Z 508.841,A -85,B 0,C 180,E1 -14663.969,E2 -14663.969} C_VEL
LIN {X 0,Y 334.154,Z 510.663,A -85,B 0,C 180,E1 -14665.174,E2 -14665.174} C_VEL
LIN {X 0,Y 333.902,Z 512.036,A -85,B 0,C 180,E1 -14666.38,E2 -14666.38} C_VEL
LIN {X 0,Y 333.912,Z 513.57,A -85,B 0,C 180,E1 -14668.794,E2 -14668.794} C_VEL
LIN {X 0,Y 333.906,Z 513.794,A -85,B 0,C 180,E1 -14670,E2 -14670} C_VEL
LIN {X 0,Y 333.912,Z 513.61,A -85,B 0,C 180,E1 -14671.206,E2 -14671.206} C_VEL
LIN {X 0,Y 333.894,Z 512.129,A -85,B 0,C 180,E1 -14673.62,E2 -14673.62} C_VEL
LIN {X 0,Y 334.142,Z 510.798,A -85,B 0,C 180,E1 -14674.826,E2 -14674.826} C_VEL
LIN {X 0,Y 334.668,Z 507.98,A -85,B 0,C 180,E1 -14676.632,E2 -14676.632} C_VEL
LIN {X 0,Y 335.331,Z 504.162,A -85,B 0,C 180,E1 -14678.436,E2 -14678.436} C_VEL
LIN {X 0,Y 336.012,Z 498.261,A -85,B 0,C 180,E1 -14680.563,E2 -14680.563} C_VEL
LIN {X 0,Y 337.039,Z 491.858,A -85,B 0,C 180,E1 -14682.341,E2 -14682.341} C_VEL
LIN {X 0,Y 338.239,Z 483.823,A -85,B 0,C 180,E1 -14684.131,E2 -14684.131} C_VEL
LIN {X 0,Y 339.197,Z 475.605,A -85,B 0,C 180,E1 -14685.626,E2 -14685.626} C_VEL
LIN {X 0,Y 340.372,Z 465.412,A -85,B 0,C 180,E1 -14687.112,E2 -14687.112} C_VEL
LIN {X 0,Y 341.551,Z 454.427,A -85,B 0,C 180,E1 -14688.383,E2 -14688.383} C_VEL
LIN {X 0,Y 338.74,Z 444.568,A -85,B 0,C 180,E1 -14689.562,E2 -14689.562} C_VEL
LIN {X 0,Y 334.842,Z 433.238,A -85,B 0,C 180,E1 -14690.725,E2 -14690.725} C_VEL
LIN {X 0,Y 333.759,Z 429.913,A -85,B 0,C 180,E1 -14691.051,E2 -14691.051} C_VEL
LIN {X 0,Y 333.722,Z 429.917,A -85,B 0,C 180,E1 -14695.101,E2 -14695.101} C_VEL
LIN {X 0,Y 333.719,Z 429.911,A -85,B 0,C 180,E1 -14697.809,E2 -14697.809} C_VEL
LIN {X 0,Y 333.692,Z 429.915,A -85,B 0,C 180,E1 -14700.363,E2 -14700.363} C_VEL
LIN {X 0,Y 333.677,Z 429.919,A -85,B 0,C 180,E1 -14704.658,E2 -14704.658} C_VEL
LIN {X 0,Y 333.662,Z 429.921,A -85,B 0,C 180,E1 -14707.65,E2 -14707.65} C_VEL
LIN {X 0,Y 333.701,Z 429.918,A -85,B 0,C 180,E1 -14710.759,E2 -14710.759} C_VEL
LIN {X 0,Y 333.671,Z 429.919,A -85,B 0,C 180,E1 -14714.264,E2 -14714.264} C_VEL
LIN {X 0,Y 333.645,Z 429.922,A -85,B 0,C 180,E1 -14717.619,E2 -14717.619} C_VEL
LIN {X 0,Y 333.654,Z 429.924,A -85,B 0,C 180,E1 -14721.202,E2 -14721.202} C_VEL
LIN {X 0,Y 333.675,Z 429.919,A -85,B 0,C 180,E1 -14725.046,E2 -14725.046} C_VEL
LIN {X 0,Y 333.632,Z 429.923,A -85,B 0,C 180,E1 -14728.222,E2 -14728.222} C_VEL
LIN {X 0,Y 333.673,Z 429.917,A -85,B 0,C 180,E1 -14730.271,E2 -14730.271} C_VEL
LIN {X 0,Y 333.004,Z 430.004,A -85,B 0,C 180,E1 -14731.278,E2 -14731.278} C_VEL
LIN {X 0,Y 330.155,Z 430.36,A -85,B 0,C 180,E1 -14732.918,E2 -14732.918} C_VEL
LIN {X 0,Y 327.75,Z 430.657,A -85,B 0,C 180,E1 -14734.245,E2 -14734.245} C_VEL
LIN {X 0,Y 326.727,Z 430.785,A -85,B 0,C 180,E1 -14735.273,E2 -14735.273} C_VEL
LIN {X 0,Y 326.649,Z 430.793,A -85,B 0,C 180,E1 -14735.621,E2 -14735.621} C_VEL
LIN {X 0,Y 326.65,Z 430.796,A -85,B 0,C 180,E1 -14738.545,E2 -14738.545} C_VEL
LIN {X 0,Y 326.746,Z 430.782,A -85,B 0,C 180,E1 -14741.177,E2 -14741.177} C_VEL
LIN {X 0,Y 326.765,Z 430.779,A -85,B 0,C 180,E1 -14745.433,E2 -14745.433} C_VEL
LIN {X 0,Y 326.775,Z 430.78,A -85,B 0,C 180,E1 -14748.839,E2 -14748.839} C_VEL
LIN {X 0,Y 326.947,Z 430.76,A -85,B 0,C 180,E1 -14752.59,E2 -14752.59} C_VEL
LIN {X 0,Y 326.987,Z 430.75,A -85,B 0,C 180,E1 -14753.831,E2 -14753.831} C_VEL
LIN {X 0,Y 327.05,Z 430.743,A -85,B 0,C 180,E1 -14757.537,E2 -14757.537} C_VEL
LIN {X 0,Y 327.22,Z 430.724,A -85,B 0,C 180,E1 -14760,E2 -14760} C_VEL
LIN {X 0,Y 327.051,Z 430.747,A -85,B 0,C 180,E1 -14762.463,E2 -14762.463} C_VEL
LIN {X 0,Y 326.986,Z 430.755,A -85,B 0,C 180,E1 -14766.169,E2 -14766.169} C_VEL
LIN {X 0,Y 326.807,Z 430.775,A -85,B 0,C 180,E1 -14769.906,E2 -14769.906} C_VEL
LIN {X 0,Y 326.762,Z 430.779,A -85,B 0,C 180,E1 -14773.685,E2 -14773.685} C_VEL
LIN {X 0,Y 326.701,Z 430.786,A -85,B 0,C 180,E1 -14777.528,E2 -14777.528} C_VEL
LIN {X 0,Y 326.662,Z 430.797,A -85,B 0,C 180,E1 -14780.135,E2 -14780.135} C_VEL
LIN {X 0,Y 326.65,Z 430.799,A -85,B 0,C 180,E1 -14784.129,E2 -14784.129} C_VEL
LIN {X 0,Y 326.685,Z 430.789,A -85,B 0,C 180,E1 -14786.858,E2 -14786.858} C_VEL
LIN {X 0,Y 326.635,Z 430.797,A -85,B 0,C 180,E1 -14790.61,E2 -14790.61} C_VEL
LIN {X 0,Y 326.609,Z 430.803,A -85,B 0,C 180,E1 -14794.019,E2 -14794.019} C_VEL
LIN {X 0,Y 326.629,Z 430.797,A -85,B 0,C 180,E1 -14797.239,E2 -14797.239} C_VEL
LIN {X 0,Y 326.579,Z 430.807,A -85,B 0,C 180,E1 -14801.131,E2 -14801.131} C_VEL
LIN {X 0,Y 326.591,Z 430.814,A -85,B 0,C 180,E1 -14802.157,E2 -14802.157} C_VEL
LIN {X 0,Y 328.216,Z 438.694,A -85,B 0,C 180,E1 -14805.834,E2 -14805.834} C_VEL
LIN {X 0,Y 329.817,Z 446.474,A -85,B 0,C 180,E1 -14809.225,E2 -14809.225} C_VEL
LIN {X 0,Y 330.899,Z 453.204,A -85,B 0,C 180,E1 -14811.98,E2 -14811.98} C_VEL
LIN {X 0,Y 329.631,Z 462.938,A -85,B 0,C 180,E1 -14815.598,E2 -14815.598} C_VEL
LIN {X 0,Y 328.549,Z 471.813,A -85,B 0,C 180,E1 -14818.831,E2 -14818.831} C_VEL
LIN {X 0,Y 327.483,Z 482.035,A -85,B 0,C 180,E1 -14822.522,E2 -14822.522} C_VEL
LIN {X 0,Y 326.685,Z 491.334,A -85,B 0,C 180,E1 -14825.874,E2 -14825.874} C_VEL
LIN {X 0,Y 326.336,Z 496.079,A -85,B 0,C 180,E1 -14827.592,E2 -14827.592} C_VEL
LIN {X 0,Y 328.495,Z 510.694,A -85,B 0,C 180,E1 -14828.274,E2 -14828.274} C_VEL
LIN {X 0,Y 329.631,Z 523.189,A -85,B 0,C 180,E1 -14829.053,E2 -14829.053} C_VEL
LIN {X 0,Y 330.213,Z 536.079,A -85,B 0,C 180,E1 -14830.091,E2 -14830.091} C_VEL
LIN {X 0,Y 330.218,Z 547.389,A -85,B 0,C 180,E1 -14831.222,E2 -14831.222} C_VEL
LIN {X 0,Y 330.049,Z 554.148,A -85,B 0,C 180,E1 -14832.015,E2 -14832.015} C_VEL
LIN {X 0,Y 328.785,Z 564.198,A -85,B 0,C 180,E1 -14833.387,E2 -14833.387} C_VEL
LIN {X 0,Y 327.437,Z 574.186,A -85,B 0,C 180,E1 -14835.074,E2 -14835.074} C_VEL
LIN {X 0,Y 326.646,Z 581.669,A -85,B 0,C 180,E1 -14836.627,E2 -14836.627} C_VEL
LIN {X 0,Y 325.983,Z 589.073,A -85,B 0,C 180,E1 -14838.497,E2 -14838.497} C_VEL
LIN {X 0,Y 325.612,Z 595.867,A -85,B 0,C 180,E1 -14840.684,E2 -14840.684} C_VEL
LIN {X 0,Y 325.6,Z 600.402,A -85,B 0,C 180,E1 -14842.559,E2 -14842.559} C_VEL
LIN {X 0,Y 325.698,Z 602.819,A -85,B 0,C 180,E1 -14843.806,E2 -14843.806} C_VEL
LIN {X 0,Y 325.906,Z 604.797,A -85,B 0,C 180,E1 -14845.052,E2 -14845.052} C_VEL
LIN {X 0,Y 326.05,Z 606.28,A -85,B 0,C 180,E1 -14846.292,E2 -14846.292} C_VEL
LIN {X 0,Y 326.13,Z 607.334,A -85,B 0,C 180,E1 -14847.53,E2 -14847.53} C_VEL
LIN {X 0,Y 326.538,Z 608.252,A -85,B 0,C 180,E1 -14850,E2 -14850} C_VEL
LIN {X 0,Y 326.131,Z 607.327,A -85,B 0,C 180,E1 -14852.47,E2 -14852.47} C_VEL
LIN {X 0,Y 326.05,Z 606.27,A -85,B 0,C 180,E1 -14853.708,E2 -14853.708} C_VEL
LIN {X 0,Y 325.905,Z 604.782,A -85,B 0,C 180,E1 -14854.949,E2 -14854.949} C_VEL
LIN {X 0,Y 325.623,Z 601.574,A -85,B 0,C 180,E1 -14856.865,E2 -14856.865} C_VEL
LIN {X 0,Y 325.596,Z 597.495,A -85,B 0,C 180,E1 -14858.691,E2 -14858.691} C_VEL
LIN {X 0,Y 325.803,Z 591.127,A -85,B 0,C 180,E1 -14860.88,E2 -14860.88} C_VEL
LIN {X 0,Y 326.394,Z 584.239,A -85,B 0,C 180,E1 -14862.751,E2 -14862.751} C_VEL
LIN {X 0,Y 327.108,Z 577.413,A -85,B 0,C 180,E1 -14864.274,E2 -14864.274} C_VEL
LIN {X 0,Y 327.935,Z 570.734,A -85,B 0,C 180,E1 -14865.538,E2 -14865.538} C_VEL
LIN {X 0,Y 329.074,Z 560.926,A -85,B 0,C 180,E1 -14867.077,E2 -14867.077} C_VEL
LIN {X 0,Y 330.18,Z 551.399,A -85,B 0,C 180,E1 -14868.298,E2 -14868.298} C_VEL
LIN {X 0,Y 330.25,Z 539.458,A -85,B 0,C 180,E1 -14869.583,E2 -14869.583} C_VEL
LIN {X 0,Y 329.951,Z 528.39,A -85,B 0,C 180,E1 -14870.542,E2 -14870.542} C_VEL
LIN {X 0,Y 328.939,Z 514.937,A -85,B 0,C 180,E1 -14871.463,E2 -14871.463} C_VEL
LIN {X 0,Y 327.008,Z 500.864,A -85,B 0,C 180,E1 -14872.198,E2 -14872.198} C_VEL
LIN {X 0,Y 326.3,Z 496.032,A -85,B 0,C 180,E1 -14872.407,E2 -14872.407} C_VEL
LIN {X 0,Y 327.151,Z 485.717,A -85,B 0,C 180,E1 -14876.128,E2 -14876.128} C_VEL
LIN {X 0,Y 328.229,Z 474.381,A -85,B 0,C 180,E1 -14880.211,E2 -14880.211} C_VEL
LIN {X 0,Y 329.373,Z 464.792,A -85,B 0,C 180,E1 -14883.696,E2 -14883.696} C_VEL
LIN {X 0,Y 330.676,Z 455.1,A -85,B 0,C 180,E1 -14887.281,E2 -14887.281} C_VEL
LIN {X 0,Y 330.827,Z 452.725,A -85,B 0,C 180,E1 -14888.185,E2 -14888.185} C_VEL
LIN {X 0,Y 329.802,Z 446.413,A -85,B 0,C 180,E1 -14890.773,E2 -14890.773} C_VEL
LIN {X 0,Y 328.21,Z 438.611,A -85,B 0,C 180,E1 -14894.165,E2 -14894.165} C_VEL
LIN {X 0,Y 326.592,Z 430.807,A -85,B 0,C 180,E1 -14897.843,E2 -14897.843} C_VEL
LIN {X 0,Y 326.626,Z 430.8,A -85,B 0,C 180,E1 -14901.392,E2 -14901.392} C_VEL
LIN {X 0,Y 326.622,Z 430.797,A -85,B 0,C 180,E1 -14904.851,E2 -14904.851} C_VEL
LIN {X 0,Y 326.612,Z 430.799,A -85,B 0,C 180,E1 -14907.456,E2 -14907.456} C_VEL
LIN {X 0,Y 326.65,Z 430.797,A -85,B 0,C 180,E1 -14910.34,E2 -14910.34} C_VEL
LIN {X 0,Y 326.692,Z 430.789,A -85,B 0,C 180,E1 -14914.516,E2 -14914.516} C_VEL
LIN {X 0,Y 326.623,Z 430.797,A -85,B 0,C 180,E1 -14918.544,E2 -14918.544} C_VEL
LIN {X 0,Y 326.747,Z 430.782,A -85,B 0,C 180,E1 -14921.178,E2 -14921.178} C_VEL
LIN {X 0,Y 326.766,Z 430.782,A -85,B 0,C 180,E1 -14925.433,E2 -14925.433} C_VEL
LIN {X 0,Y 326.775,Z 430.778,A -85,B 0,C 180,E1 -14928.839,E2 -14928.839} C_VEL
LIN {X 0,Y 326.946,Z 430.757,A -85,B 0,C 180,E1 -14932.59,E2 -14932.59} C_VEL
LIN {X 0,Y 326.987,Z 430.756,A -85,B 0,C 180,E1 -14933.831,E2 -14933.831} C_VEL
LIN {X 0,Y 327.052,Z 430.748,A -85,B 0,C 180,E1 -14937.537,E2 -14937.537} C_VEL
LIN {X 0,Y 327.221,Z 430.724,A -85,B 0,C 180,E1 -14940,E2 -14940} C_VEL
LIN {X 0,Y 327.05,Z 430.743,A -85,B 0,C 180,E1 -14942.463,E2 -14942.463} C_VEL
LIN {X 0,Y 326.954,Z 430.755,A -85,B 0,C 180,E1 -14946.616,E2 -14946.616} C_VEL
LIN {X 0,Y 326.809,Z 430.775,A -85,B 0,C 180,E1 -14949.907,E2 -14949.907} C_VEL
LIN {X 0,Y 326.764,Z 430.775,A -85,B 0,C 180,E1 -14953.685,E2 -14953.685} C_VEL
LIN {X 0,Y 326.703,Z 430.785,A -85,B 0,C 180,E1 -14957.528,E2 -14957.528} C_VEL
LIN {X 0,Y 326.669,Z 430.79,A -85,B 0,C 180,E1 -14960.135,E2 -14960.135} C_VEL
LIN {X 0,Y 326.656,Z 430.79,A -85,B 0,C 180,E1 -14964.129,E2 -14964.129} C_VEL
LIN {X 0,Y 326.686,Z 430.785,A -85,B 0,C 180,E1 -14966.858,E2 -14966.858} C_VEL
LIN {X 0,Y 326.637,Z 430.793,A -85,B 0,C 180,E1 -14970.61,E2 -14970.61} C_VEL
LIN {X 0,Y 326.61,Z 430.798,A -85,B 0,C 180,E1 -14974.019,E2 -14974.019} C_VEL
LIN {X 0,Y 326.63,Z 430.801,A -85,B 0,C 180,E1 -14977.239,E2 -14977.239} C_VEL
LIN {X 0,Y 326.581,Z 430.807,A -85,B 0,C 180,E1 -14981.131,E2 -14981.131} C_VEL
LIN {X 0,Y 326.586,Z 430.803,A -85,B 0,C 180,E1 -14984.753,E2 -14984.753} C_VEL
LIN {X 0,Y 326.625,Z 430.795,A -85,B 0,C 180,E1 -14988.162,E2 -14988.162} C_VEL
LIN {X 0,Y 326.651,Z 430.794,A -85,B 0,C 180,E1 -14991.395,E2 -14991.395} C_VEL
LIN {X 0,Y 326.623,Z 430.8,A -85,B 0,C 180,E1 -14994.851,E2 -14994.851} C_VEL
LIN {X 0,Y 326.61,Z 430.799,A -85,B 0,C 180,E1 -14997.456,E2 -14997.456} C_VEL
LIN {X 0,Y 326.65,Z 430.794,A -85,B 0,C 180,E1 -15000.34,E2 -15000.34} C_VEL
LIN {X 0,Y 326.693,Z 430.792,A -85,B 0,C 180,E1 -15004.516,E2 -15004.516} C_VEL
LIN {X 0,Y 326.653,Z 430.846,A -85,B 0,C 180,E1 -15008.607,E2 -15008.607} C_VEL
LIN {X 0,Y 330.633,Z 441.826,A -85,B 0,C 180,E1 -15009.708,E2 -15009.708} C_VEL
LIN {X 0,Y 333.937,Z 452.807,A -85,B 0,C 180,E1 -15010.99,E2 -15010.99} C_VEL
LIN {X 0,Y 334.666,Z 455.459,A -85,B 0,C 180,E1 -15011.333,E2 -15011.333} C_VEL
LIN {X 0,Y 333.745,Z 465.613,A -85,B 0,C 180,E1 -15012.538,E2 -15012.538} C_VEL
LIN {X 0,Y 332.531,Z 475.959,A -85,B 0,C 180,E1 -15014.053,E2 -15014.053} C_VEL
LIN {X 0,Y 331.471,Z 484.32,A -85,B 0,C 180,E1 -15015.574,E2 -15015.574} C_VEL
LIN {X 0,Y 330.182,Z 492.449,A -85,B 0,C 180,E1 -15017.398,E2 -15017.398} C_VEL
LIN {X 0,Y 329.223,Z 498.571,A -85,B 0,C 180,E1 -15019.106,E2 -15019.106} C_VEL
LIN {X 0,Y 328.622,Z 503.367,A -85,B 0,C 180,E1 -15020.77,E2 -15020.77} C_VEL
LIN {X 0,Y 327.833,Z 507.612,A -85,B 0,C 180,E1 -15022.61,E2 -15022.61} C_VEL
LIN {X 0,Y 327.468,Z 509.847,A -85,B 0,C 180,E1 -15023.84,E2 -15023.84} C_VEL
LIN {X 0,Y 327.151,Z 511.669,A -85,B 0,C 180,E1 -15025.07,E2 -15025.07} C_VEL
LIN {X 0,Y 326.888,Z 513.042,A -85,B 0,C 180,E1 -15026.302,E2 -15026.302} C_VEL
LIN {X 0,Y 326.892,Z 514.574,A -85,B 0,C 180,E1 -15028.768,E2 -15028.768} C_VEL
LIN {X 0,Y 326.884,Z 514.798,A -85,B 0,C 180,E1 -15030,E2 -15030} C_VEL
LIN {X 0,Y 326.892,Z 514.614,A -85,B 0,C 180,E1 -15031.232,E2 -15031.232} C_VEL
LIN {X 0,Y 326.88,Z 513.134,A -85,B 0,C 180,E1 -15033.698,E2 -15033.698} C_VEL
LIN {X 0,Y 327.139,Z 511.803,A -85,B 0,C 180,E1 -15034.93,E2 -15034.93} C_VEL
LIN {X 0,Y 327.69,Z 508.984,A -85,B 0,C 180,E1 -15036.774,E2 -15036.774} C_VEL
LIN {X 0,Y 328.381,Z 505.166,A -85,B 0,C 180,E1 -15038.616,E2 -15038.616} C_VEL
LIN {X 0,Y 329.105,Z 499.267,A -85,B 0,C 180,E1 -15040.787,E2 -15040.787} C_VEL
LIN {X 0,Y 330.178,Z 492.861,A -85,B 0,C 180,E1 -15042.602,E2 -15042.602} C_VEL
LIN {X 0,Y 331.428,Z 484.825,A -85,B 0,C 180,E1 -15044.428,E2 -15044.428} C_VEL
LIN {X 0,Y 332.434,Z 476.607,A -85,B 0,C 180,E1 -15045.952,E2 -15045.952} C_VEL
LIN {X 0,Y 333.662,Z 466.413,A -85,B 0,C 180,E1 -15047.467,E2 -15047.467} C_VEL
LIN {X 0,Y 334.796,Z 456.319,A -85,B 0,C 180,E1 -15048.667,E2 -15048.667} C_VEL
LIN {X 0,Y 331.769,Z 445.41,A -85,B 0,C 180,E1 -15050.011,E2 -15050.011} C_VEL
LIN {X 0,Y 327.946,Z 434.387,A -85,B 0,C 180,E1 -15051.175,E2 -15051.175} C_VEL
LIN {X 0,Y 326.686,Z 430.794,A -85,B 0,C 180,E1 -15051.513,E2 -15051.513} C_VEL
LIN {X 0,Y 326.692,Z 430.792,A -85,B 0,C 180,E1 -15055.484,E2 -15055.484} C_VEL
LIN {X 0,Y 326.65,Z 430.794,A -85,B 0,C 180,E1 -15059.66,E2 -15059.66} C_VEL
LIN {X 0,Y 326.621,Z 430.799,A -85,B 0,C 180,E1 -15062.946,E2 -15062.946} C_VEL
LIN {X 0,Y 326.616,Z 430.8,A -85,B 0,C 180,E1 -15065.519,E2 -15065.519} C_VEL
LIN {X 0,Y 326.65,Z 430.798,A -85,B 0,C 180,E1 -15069.235,E2 -15069.235} C_VEL
LIN {X 0,Y 326.63,Z 430.801,A -85,B 0,C 180,E1 -15072.982,E2 -15072.982} C_VEL
LIN {X 0,Y 326.588,Z 430.806,A -85,B 0,C 180,E1 -15077.026,E2 -15077.026} C_VEL
LIN {X 0,Y 326.613,Z 430.802,A -85,B 0,C 180,E1 -15080.773,E2 -15080.773} C_VEL
LIN {X 0,Y 326.614,Z 430.799,A -85,B 0,C 180,E1 -15084.48,E2 -15084.48} C_VEL
LIN {X 0,Y 326.609,Z 430.798,A -85,B 0,C 180,E1 -15087.455,E2 -15087.455} C_VEL
LIN {X 0,Y 326.649,Z 430.795,A -85,B 0,C 180,E1 -15090.34,E2 -15090.34} C_VEL
LIN {X 0,Y 326.692,Z 430.791,A -85,B 0,C 180,E1 -15094.516,E2 -15094.516} C_VEL
LIN {X 0,Y 326.649,Z 430.793,A -85,B 0,C 180,E1 -15095.621,E2 -15095.621} C_VEL
LIN {X 0,Y 326.012,Z 430.877,A -85,B 0,C 180,E1 -15096.65,E2 -15096.65} C_VEL
LIN {X 0,Y 323.229,Z 431.226,A -85,B 0,C 180,E1 -15098.325,E2 -15098.325} C_VEL
LIN {X 0,Y 320.839,Z 431.524,A -85,B 0,C 180,E1 -15099.682,E2 -15099.682} C_VEL
LIN {X 0,Y 319.783,Z 431.653,A -85,B 0,C 180,E1 -15100.731,E2 -15100.731} C_VEL
LIN {X 0,Y 319.681,Z 431.662,A -85,B 0,C 180,E1 -15101.087,E2 -15101.087} C_VEL
LIN {X 0,Y 319.733,Z 431.655,A -85,B 0,C 180,E1 -15105.276,E2 -15105.276} C_VEL
LIN {X 0,Y 319.755,Z 431.652,A -85,B 0,C 180,E1 -15109.873,E2 -15109.873} C_VEL
LIN {X 0,Y 319.94,Z 431.627,A -85,B 0,C 180,E1 -15113.694,E2 -15113.694} C_VEL
LIN {X 0,Y 319.994,Z 431.622,A -85,B 0,C 180,E1 -15117.482,E2 -15117.482} C_VEL
LIN {X 0,Y 320.171,Z 431.602,A -85,B 0,C 180,E1 -15120,E2 -15120} C_VEL
LIN {X 0,Y 319.995,Z 431.625,A -85,B 0,C 180,E1 -15122.518,E2 -15122.518} C_VEL
LIN {X 0,Y 319.94,Z 431.633,A -85,B 0,C 180,E1 -15126.306,E2 -15126.306} C_VEL
LIN {X 0,Y 319.755,Z 431.656,A -85,B 0,C 180,E1 -15130.127,E2 -15130.127} C_VEL
LIN {X 0,Y 319.733,Z 431.656,A -85,B 0,C 180,E1 -15134.724,E2 -15134.724} C_VEL
LIN {X 0,Y 319.69,Z 431.661,A -85,B 0,C 180,E1 -15139.038,E2 -15139.038} C_VEL
LIN {X 0,Y 319.562,Z 431.677,A -85,B 0,C 180,E1 -15143.32,E2 -15143.32} C_VEL
LIN {X 0,Y 319.636,Z 431.672,A -85,B 0,C 180,E1 -15146.088,E2 -15146.088} C_VEL
LIN {X 0,Y 319.581,Z 431.674,A -85,B 0,C 180,E1 -15148.934,E2 -15148.934} C_VEL
LIN {X 0,Y 319.533,Z 431.684,A -85,B 0,C 180,E1 -15151.862,E2 -15151.862} C_VEL
LIN {X 0,Y 319.582,Z 431.677,A -85,B 0,C 180,E1 -15155.543,E2 -15155.543} C_VEL
LIN {X 0,Y 319.574,Z 431.679,A -85,B 0,C 180,E1 -15158.008,E2 -15158.008} C_VEL
LIN {X 0,Y 319.567,Z 431.85,A -85,B 0,C 180,E1 -15161.72,E2 -15161.72} C_VEL
LIN {X 0,Y 321.215,Z 439.854,A -85,B 0,C 180,E1 -15165.562,E2 -15165.562} C_VEL
LIN {X 0,Y 322.9,Z 448.093,A -85,B 0,C 180,E1 -15169.235,E2 -15169.235} C_VEL
LIN {X 0,Y 323.78,Z 453.198,A -85,B 0,C 180,E1 -15171.391,E2 -15171.391} C_VEL
LIN {X 0,Y 323.716,Z 456.159,A -85,B 0,C 180,E1 -15172.563,E2 -15172.563} C_VEL
LIN {X 0,Y 322.167,Z 467.748,A -85,B 0,C 180,E1 -15176.95,E2 -15176.95} C_VEL
LIN {X 0,Y 320.752,Z 479.236,A -85,B 0,C 180,E1 -15181.216,E2 -15181.216} C_VEL
LIN {X 0,Y 319.747,Z 490.303,A -85,B 0,C 180,E1 -15185.316,E2 -15185.316} C_VEL
LIN {X 0,Y 319.338,Z 494.989,A -85,B 0,C 180,E1 -15187.061,E2 -15187.061} C_VEL
LIN {X 0,Y 321.593,Z 510.41,A -85,B 0,C 180,E1 -15187.819,E2 -15187.819} C_VEL
LIN {X 0,Y 322.71,Z 522.196,A -85,B 0,C 180,E1 -15188.586,E2 -15188.586} C_VEL
LIN {X 0,Y 323.3,Z 535.031,A -85,B 0,C 180,E1 -15189.646,E2 -15189.646} C_VEL
LIN {X 0,Y 323.299,Z 546.346,A -85,B 0,C 180,E1 -15190.804,E2 -15190.804} C_VEL
LIN {X 0,Y 323.085,Z 554.32,A -85,B 0,C 180,E1 -15191.778,E2 -15191.778} C_VEL
LIN {X 0,Y 321.779,Z 564.168,A -85,B 0,C 180,E1 -15193.178,E2 -15193.178} C_VEL
LIN {X 0,Y 320.565,Z 573.17,A -85,B 0,C 180,E1 -15194.747,E2 -15194.747} C_VEL
LIN {X 0,Y 319.709,Z 580.65,A -85,B 0,C 180,E1 -15196.331,E2 -15196.331} C_VEL
LIN {X 0,Y 318.957,Z 588.049,A -85,B 0,C 180,E1 -15198.24,E2 -15198.24} C_VEL
LIN {X 0,Y 318.562,Z 594.846,A -85,B 0,C 180,E1 -15200.476,E2 -15200.476} C_VEL
LIN {X 0,Y 318.519,Z 599.381,A -85,B 0,C 180,E1 -15202.392,E2 -15202.392} C_VEL
LIN {X 0,Y 318.63,Z 601.803,A -85,B 0,C 180,E1 -15203.668,E2 -15203.668} C_VEL
LIN {X 0,Y 318.826,Z 603.781,A -85,B 0,C 180,E1 -15204.942,E2 -15204.942} C_VEL
LIN {X 0,Y 319.002,Z 605.27,A -85,B 0,C 180,E1 -15206.21,E2 -15206.21} C_VEL
LIN {X 0,Y 319.084,Z 606.326,A -85,B 0,C 180,E1 -15207.475,E2 -15207.475} C_VEL
LIN {X 0,Y 319.509,Z 607.247,A -85,B 0,C 180,E1 -15210,E2 -15210} C_VEL
LIN {X 0,Y 319.084,Z 606.318,A -85,B 0,C 180,E1 -15212.525,E2 -15212.525} C_VEL
LIN {X 0,Y 319.002,Z 605.26,A -85,B 0,C 180,E1 -15213.79,E2 -15213.79} C_VEL
LIN {X 0,Y 318.825,Z 603.765,A -85,B 0,C 180,E1 -15215.059,E2 -15215.059} C_VEL
LIN {X 0,Y 318.554,Z 600.806,A -85,B 0,C 180,E1 -15216.878,E2 -15216.878} C_VEL
LIN {X 0,Y 318.519,Z 596.47,A -85,B 0,C 180,E1 -15218.885,E2 -15218.885} C_VEL
LIN {X 0,Y 318.78,Z 590.102,A -85,B 0,C 180,E1 -15221.123,E2 -15221.123} C_VEL
LIN {X 0,Y 319.391,Z 583.21,A -85,B 0,C 180,E1 -15223.035,E2 -15223.035} C_VEL
LIN {X 0,Y 320.05,Z 576.783,A -85,B 0,C 180,E1 -15224.509,E2 -15224.509} C_VEL
LIN {X 0,Y 321.329,Z 567.893,A -85,B 0,C 180,E1 -15226.193,E2 -15226.193} C_VEL
LIN {X 0,Y 322.516,Z 558.832,A -85,B 0,C 180,E1 -15227.599,E2 -15227.599} C_VEL
LIN {X 0,Y 323.215,Z 551.678,A -85,B 0,C 180,E1 -15228.543,E2 -15228.543} C_VEL
LIN {X 0,Y 323.339,Z 540.03,A -85,B 0,C 180,E1 -15229.854,E2 -15229.854} C_VEL
LIN {X 0,Y 323.033,Z 527.376,A -85,B 0,C 180,E1 -15230.999,E2 -15230.999} C_VEL
LIN {X 0,Y 322.066,Z 514.202,A -85,B 0,C 180,E1 -15231.926,E2 -15231.926} C_VEL
LIN {X 0,Y 320.081,Z 500.083,A -85,B 0,C 180,E1 -15232.693,E2 -15232.693} C_VEL
LIN {X 0,Y 319.327,Z 494.941,A -85,B 0,C 180,E1 -15232.934,E2 -15232.934} C_VEL
LIN {X 0,Y 320.189,Z 484.694,A -85,B 0,C 180,E1 -15236.742,E2 -15236.742} C_VEL
LIN {X 0,Y 321.362,Z 473.516,A -85,B 0,C 180,E1 -15240.879,E2 -15240.879} C_VEL
LIN {X 0,Y 322.447,Z 464.92,A -85,B 0,C 180,E1 -15244.081,E2 -15244.081} C_VEL
LIN {X 0,Y 323.723,Z 456.092,A -85,B 0,C 180,E1 -15247.436,E2 -15247.436} C_VEL
LIN {X 0,Y 323.645,Z 452.114,A -85,B 0,C 180,E1 -15249.031,E2 -15249.031} C_VEL
LIN {X 0,Y 322.048,Z 443.9,A -85,B 0,C 180,E1 -15252.572,E2 -15252.572} C_VEL
LIN {X 0,Y 320.348,Z 435.63,A -85,B 0,C 180,E1 -15256.384,E2 -15256.384} C_VEL
LIN {X 0,Y 319.528,Z 431.687,A -85,B 0,C 180,E1 -15258.403,E2 -15258.403} C_VEL
LIN {X 0,Y 319.58,Z 431.679,A -85,B 0,C 180,E1 -15262.344,E2 -15262.344} C_VEL
LIN {X 0,Y 319.563,Z 431.677,A -85,B 0,C 180,E1 -15265.124,E2 -15265.124} C_VEL
LIN {X 0,Y 319.569,Z 431.675,A -85,B 0,C 180,E1 -15269.059,E2 -15269.059} C_VEL
LIN {X 0,Y 319.608,Z 431.673,A -85,B 0,C 180,E1 -15272.498,E2 -15272.498} C_VEL
LIN {X 0,Y 319.605,Z 431.671,A -85,B 0,C 180,E1 -15275.304,E2 -15275.304} C_VEL
LIN {X 0,Y 319.606,Z 431.672,A -85,B 0,C 180,E1 -15279.401,E2 -15279.401} C_VEL
LIN {X 0,Y 319.661,Z 431.668,A -85,B 0,C 180,E1 -15282.073,E2 -15282.073} C_VEL
LIN {X 0,Y 319.736,Z 431.659,A -85,B 0,C 180,E1 -15286.008,E2 -15286.008} C_VEL
LIN {X 0,Y 319.756,Z 431.657,A -85,B 0,C 180,E1 -15289.873,E2 -15289.873} C_VEL
LIN {X 0,Y 319.941,Z 431.634,A -85,B 0,C 180,E1 -15293.694,E2 -15293.694} C_VEL
LIN {X 0,Y 319.996,Z 431.626,A -85,B 0,C 180,E1 -15297.482,E2 -15297.482} C_VEL
LIN {X 0,Y 320.172,Z 431.602,A -85,B 0,C 180,E1 -15300,E2 -15300} C_VEL
LIN {X 0,Y 319.994,Z 431.622,A -85,B 0,C 180,E1 -15302.518,E2 -15302.518} C_VEL
LIN {X 0,Y 319.916,Z 431.631,A -85,B 0,C 180,E1 -15306.602,E2 -15306.602} C_VEL
LIN {X 0,Y 319.756,Z 431.652,A -85,B 0,C 180,E1 -15310.127,E2 -15310.127} C_VEL
LIN {X 0,Y 319.734,Z 431.646,A -85,B 0,C 180,E1 -15314.724,E2 -15314.724} C_VEL
LIN {X 0,Y 319.692,Z 431.657,A -85,B 0,C 180,E1 -15319.038,E2 -15319.038} C_VEL
LIN {X 0,Y 319.574,Z 431.678,A -85,B 0,C 180,E1 -15323.319,E2 -15323.319} C_VEL
LIN {X 0,Y 319.621,Z 431.662,A -85,B 0,C 180,E1 -15326.089,E2 -15326.089} C_VEL
LIN {X 0,Y 319.582,Z 431.667,A -85,B 0,C 180,E1 -15328.934,E2 -15328.934} C_VEL
LIN {X 0,Y 319.533,Z 431.68,A -85,B 0,C 180,E1 -15331.862,E2 -15331.862} C_VEL
LIN {X 0,Y 319.583,Z 431.675,A -85,B 0,C 180,E1 -15335.543,E2 -15335.543} C_VEL
LIN {X 0,Y 319.561,Z 431.676,A -85,B 0,C 180,E1 -15339.669,E2 -15339.669} C_VEL
LIN {X 0,Y 319.567,Z 431.677,A -85,B 0,C 180,E1 -15343.469,E2 -15343.469} C_VEL
LIN {X 0,Y 319.606,Z 431.674,A -85,B 0,C 180,E1 -15347.025,E2 -15347.025} C_VEL
LIN {X 0,Y 319.588,Z 431.672,A -85,B 0,C 180,E1 -15350.377,E2 -15350.377} C_VEL
LIN {X 0,Y 319.563,Z 431.675,A -85,B 0,C 180,E1 -15353.573,E2 -15353.573} C_VEL
LIN {X 0,Y 319.58,Z 431.676,A -85,B 0,C 180,E1 -15356.686,E2 -15356.686} C_VEL
LIN {X 0,Y 319.587,Z 431.673,A -85,B 0,C 180,E1 -15359.616,E2 -15359.616} C_VEL
LIN {X 0,Y 319.608,Z 431.674,A -85,B 0,C 180,E1 -15362.498,E2 -15362.498} C_VEL
LIN {X 0,Y 319.608,Z 431.672,A -85,B 0,C 180,E1 -15365.304,E2 -15365.304} C_VEL
LIN {X 0,Y 319.633,Z 431.844,A -85,B 0,C 180,E1 -15368.107,E2 -15368.107} C_VEL
LIN {X 0,Y 323.922,Z 443.658,A -85,B 0,C 180,E1 -15369.337,E2 -15369.337} C_VEL
LIN {X 0,Y 327.118,Z 454.098,A -85,B 0,C 180,E1 -15370.605,E2 -15370.605} C_VEL
LIN {X 0,Y 328.012,Z 457.742,A -85,B 0,C 180,E1 -15371.09,E2 -15371.09} C_VEL
LIN {X 0,Y 326.768,Z 468.922,A -85,B 0,C 180,E1 -15372.476,E2 -15372.476} C_VEL
LIN {X 0,Y 325.581,Z 478.746,A -85,B 0,C 180,E1 -15374.025,E2 -15374.025} C_VEL
LIN {X 0,Y 324.195,Z 488.24,A -85,B 0,C 180,E1 -15375.884,E2 -15375.884} C_VEL
LIN {X 0,Y 322.943,Z 495.813,A -85,B 0,C 180,E1 -15377.75,E2 -15377.75} C_VEL
LIN {X 0,Y 322.165,Z 501.078,A -85,B 0,C 180,E1 -15379.357,E2 -15379.357} C_VEL
LIN {X 0,Y 321.473,Z 505.924,A -85,B 0,C 180,E1 -15381.197,E2 -15381.197} C_VEL
LIN {X 0,Y 320.721,Z 509.807,A -85,B 0,C 180,E1 -15383.078,E2 -15383.078} C_VEL
LIN {X 0,Y 320.149,Z 512.675,A -85,B 0,C 180,E1 -15384.962,E2 -15384.962} C_VEL
LIN {X 0,Y 319.875,Z 514.048,A -85,B 0,C 180,E1 -15386.221,E2 -15386.221} C_VEL
LIN {X 0,Y 319.872,Z 515.579,A -85,B 0,C 180,E1 -15388.741,E2 -15388.741} C_VEL
LIN {X 0,Y 319.862,Z 515.803,A -85,B 0,C 180,E1 -15390,E2 -15390} C_VEL
LIN {X 0,Y 319.871,Z 515.619,A -85,B 0,C 180,E1 -15391.259,E2 -15391.259} C_VEL
LIN {X 0,Y 319.867,Z 514.139,A -85,B 0,C 180,E1 -15393.779,E2 -15393.779} C_VEL
LIN {X 0,Y 320.137,Z 512.807,A -85,B 0,C 180,E1 -15395.038,E2 -15395.038} C_VEL
LIN {X 0,Y 320.714,Z 509.988,A -85,B 0,C 180,E1 -15396.922,E2 -15396.922} C_VEL
LIN {X 0,Y 321.434,Z 506.17,A -85,B 0,C 180,E1 -15398.804,E2 -15398.804} C_VEL
LIN {X 0,Y 322.203,Z 500.273,A -85,B 0,C 180,E1 -15401.02,E2 -15401.02} C_VEL
LIN {X 0,Y 323.323,Z 493.864,A -85,B 0,C 180,E1 -15402.874,E2 -15402.874} C_VEL
LIN {X 0,Y 324.626,Z 485.828,A -85,B 0,C 180,E1 -15404.737,E2 -15404.737} C_VEL
LIN {X 0,Y 325.682,Z 477.609,A -85,B 0,C 180,E1 -15406.292,E2 -15406.292} C_VEL
LIN {X 0,Y 326.964,Z 467.414,A -85,B 0,C 180,E1 -15407.836,E2 -15407.836} C_VEL
LIN {X 0,Y 327.994,Z 457.313,A -85,B 0,C 180,E1 -15409.072,E2 -15409.072} C_VEL
LIN {X 0,Y 325.182,Z 447.5,A -85,B 0,C 180,E1 -15410.329,E2 -15410.329} C_VEL
LIN {X 0,Y 321.557,Z 436.987,A -85,B 0,C 180,E1 -15411.5,E2 -15411.5} C_VEL
LIN {X 0,Y 319.646,Z 431.669,A -85,B 0,C 180,E1 -15412.023,E2 -15412.023} C_VEL
LIN {X 0,Y 319.636,Z 431.667,A -85,B 0,C 180,E1 -15416.088,E2 -15416.088} C_VEL
LIN {X 0,Y 319.582,Z 431.672,A -85,B 0,C 180,E1 -15418.934,E2 -15418.934} C_VEL
LIN {X 0,Y 319.534,Z 431.678,A -85,B 0,C 180,E1 -15421.862,E2 -15421.862} C_VEL
LIN {X 0,Y 319.583,Z 431.676,A -85,B 0,C 180,E1 -15425.543,E2 -15425.543} C_VEL
LIN {X 0,Y 319.604,Z 431.671,A -85,B 0,C 180,E1 -15428.004,E2 -15428.004} C_VEL
LIN {X 0,Y 319.599,Z 431.673,A -85,B 0,C 180,E1 -15431.611,E2 -15431.611} C_VEL
LIN {X 0,Y 319.566,Z 431.679,A -85,B 0,C 180,E1 -15435.271,E2 -15435.271} C_VEL
LIN {X 0,Y 319.531,Z 431.683,A -85,B 0,C 180,E1 -15438.712,E2 -15438.712} C_VEL
LIN {X 0,Y 319.556,Z 431.678,A -85,B 0,C 180,E1 -15442.349,E2 -15442.349} C_VEL
LIN {X 0,Y 319.562,Z 431.68,A -85,B 0,C 180,E1 -15445.123,E2 -15445.123} C_VEL
LIN {X 0,Y 319.568,Z 431.679,A -85,B 0,C 180,E1 -15449.059,E2 -15449.059} C_VEL
LIN {X 0,Y 319.608,Z 431.673,A -85,B 0,C 180,E1 -15452.498,E2 -15452.498} C_VEL
LIN {X 0,Y 319.583,Z 431.673,A -85,B 0,C 180,E1 -15455.607,E2 -15455.607} C_VEL
LIN {X 0,Y 319.618,Z 431.67,A -85,B 0,C 180,E1 -15459.401,E2 -15459.401} C_VEL
LIN {X 0,Y 319.681,Z 431.662,A -85,B 0,C 180,E1 -15461.087,E2 -15461.087} C_VEL
LIN {X 0,Y 318.975,Z 431.752,A -85,B 0,C 180,E1 -15462.139,E2 -15462.139} C_VEL
LIN {X 0,Y 316.129,Z 432.103,A -85,B 0,C 180,E1 -15463.852,E2 -15463.852} C_VEL
LIN {X 0,Y 313.743,Z 432.402,A -85,B 0,C 180,E1 -15465.24,E2 -15465.24} C_VEL
LIN {X 0,Y 312.721,Z 432.531,A -85,B 0,C 180,E1 -15466.315,E2 -15466.315} C_VEL
LIN {X 0,Y 312.638,Z 432.537,A -85,B 0,C 180,E1 -15466.678,E2 -15466.678} C_VEL
LIN {X 0,Y 312.757,Z 432.526,A -85,B 0,C 180,E1 -15470.95,E2 -15470.95} C_VEL
LIN {X 0,Y 312.896,Z 432.504,A -85,B 0,C 180,E1 -15473.552,E2 -15473.552} C_VEL
LIN {X 0,Y 312.94,Z 432.501,A -85,B 0,C 180,E1 -15477.426,E2 -15477.426} C_VEL
LIN {X 0,Y 313.123,Z 432.48,A -85,B 0,C 180,E1 -15480,E2 -15480} C_VEL
LIN {X 0,Y 312.941,Z 432.504,A -85,B 0,C 180,E1 -15482.574,E2 -15482.574} C_VEL
LIN {X 0,Y 312.896,Z 432.509,A -85,B 0,C 180,E1 -15486.448,E2 -15486.448} C_VEL
LIN {X 0,Y 312.701,Z 432.535,A -85,B 0,C 180,E1 -15490.358,E2 -15490.358} C_VEL
LIN {X 0,Y 312.702,Z 432.532,A -85,B 0,C 180,E1 -15494.888,E2 -15494.888} C_VEL
LIN {X 0,Y 312.631,Z 432.54,A -85,B 0,C 180,E1 -15499.236,E2 -15499.236} C_VEL
LIN {X 0,Y 312.527,Z 432.554,A -85,B 0,C 180,E1 -15502.78,E2 -15502.78} C_VEL
LIN {X 0,Y 312.604,Z 432.548,A -85,B 0,C 180,E1 -15505.935,E2 -15505.935} C_VEL
LIN {X 0,Y 312.54,Z 432.553,A -85,B 0,C 180,E1 -15509.651,E2 -15509.651} C_VEL
LIN {X 0,Y 312.521,Z 432.558,A -85,B 0,C 180,E1 -15513.689,E2 -15513.689} C_VEL
LIN {X 0,Y 312.539,Z 432.554,A -85,B 0,C 180,E1 -15517.383,E2 -15517.383} C_VEL
LIN {X 0,Y 312.503,Z 432.709,A -85,B 0,C 180,E1 -15521.182,E2 -15521.182} C_VEL
LIN {X 0,Y 314.04,Z 440.094,A -85,B 0,C 180,E1 -15524.845,E2 -15524.845} C_VEL
LIN {X 0,Y 315.654,Z 448.045,A -85,B 0,C 180,E1 -15528.516,E2 -15528.516} C_VEL
LIN {X 0,Y 316.716,Z 453.62,A -85,B 0,C 180,E1 -15530.956,E2 -15530.956} C_VEL
LIN {X 0,Y 316.743,Z 457.132,A -85,B 0,C 180,E1 -15532.398,E2 -15532.398} C_VEL
LIN {X 0,Y 315.334,Z 466.749,A -85,B 0,C 180,E1 -15536.139,E2 -15536.139} C_VEL
LIN {X 0,Y 314.093,Z 476.241,A -85,B 0,C 180,E1 -15539.771,E2 -15539.771} C_VEL
LIN {X 0,Y 312.885,Z 488.208,A -85,B 0,C 180,E1 -15544.329,E2 -15544.329} C_VEL
LIN {X 0,Y 312.374,Z 493.966,A -85,B 0,C 180,E1 -15546.531,E2 -15546.531} C_VEL
LIN {X 0,Y 314.586,Z 508.916,A -85,B 0,C 180,E1 -15547.277,E2 -15547.277} C_VEL
LIN {X 0,Y 315.845,Z 521.428,A -85,B 0,C 180,E1 -15548.117,E2 -15548.117} C_VEL
LIN {X 0,Y 316.406,Z 533.983,A -85,B 0,C 180,E1 -15549.183,E2 -15549.183} C_VEL
LIN {X 0,Y 316.386,Z 545.302,A -85,B 0,C 180,E1 -15550.368,E2 -15550.368} C_VEL
LIN {X 0,Y 316.128,Z 554.491,A -85,B 0,C 180,E1 -15551.531,E2 -15551.531} C_VEL
LIN {X 0,Y 314.892,Z 563.14,A -85,B 0,C 180,E1 -15552.799,E2 -15552.799} C_VEL
LIN {X 0,Y 313.608,Z 572.66,A -85,B 0,C 180,E1 -15554.502,E2 -15554.502} C_VEL
LIN {X 0,Y 312.559,Z 580.981,A -85,B 0,C 180,E1 -15556.344,E2 -15556.344} C_VEL
LIN {X 0,Y 311.836,Z 588.084,A -85,B 0,C 180,E1 -15558.297,E2 -15558.297} C_VEL
LIN {X 0,Y 311.502,Z 593.823,A -85,B 0,C 180,E1 -15560.258,E2 -15560.258} C_VEL
LIN {X 0,Y 311.467,Z 598.365,A -85,B 0,C 180,E1 -15562.219,E2 -15562.219} C_VEL
LIN {X 0,Y 311.561,Z 600.786,A -85,B 0,C 180,E1 -15563.524,E2 -15563.524} C_VEL
LIN {X 0,Y 311.75,Z 602.766,A -85,B 0,C 180,E1 -15564.826,E2 -15564.826} C_VEL
LIN {X 0,Y 311.953,Z 604.26,A -85,B 0,C 180,E1 -15566.125,E2 -15566.125} C_VEL
LIN {X 0,Y 312.037,Z 605.317,A -85,B 0,C 180,E1 -15567.418,E2 -15567.418} C_VEL
LIN {X 0,Y 312.478,Z 606.241,A -85,B 0,C 180,E1 -15570,E2 -15570} C_VEL
LIN {X 0,Y 312.037,Z 605.309,A -85,B 0,C 180,E1 -15572.582,E2 -15572.582} C_VEL
LIN {X 0,Y 311.953,Z 604.249,A -85,B 0,C 180,E1 -15573.876,E2 -15573.876} C_VEL
LIN {X 0,Y 311.749,Z 602.748,A -85,B 0,C 180,E1 -15575.174,E2 -15575.174} C_VEL
LIN {X 0,Y 311.499,Z 599.995,A -85,B 0,C 180,E1 -15576.916,E2 -15576.916} C_VEL
LIN {X 0,Y 311.467,Z 595.448,A -85,B 0,C 180,E1 -15579.088,E2 -15579.088} C_VEL
LIN {X 0,Y 311.746,Z 589.075,A -85,B 0,C 180,E1 -15581.377,E2 -15581.377} C_VEL
LIN {X 0,Y 312.384,Z 582.179,A -85,B 0,C 180,E1 -15583.333,E2 -15583.333} C_VEL
LIN {X 0,Y 313.005,Z 576.606,A -85,B 0,C 180,E1 -15584.657,E2 -15584.657} C_VEL
LIN {X 0,Y 314.2,Z 568.683,A -85,B 0,C 180,E1 -15586.236,E2 -15586.236} C_VEL
LIN {X 0,Y 315.554,Z 558.893,A -85,B 0,C 180,E1 -15587.833,E2 -15587.833} C_VEL
LIN {X 0,Y 316.271,Z 550.625,A -85,B 0,C 180,E1 -15588.965,E2 -15588.965} C_VEL
LIN {X 0,Y 316.445,Z 538.975,A -85,B 0,C 180,E1 -15590.305,E2 -15590.305} C_VEL
LIN {X 0,Y 316.142,Z 527.133,A -85,B 0,C 180,E1 -15591.411,E2 -15591.411} C_VEL
LIN {X 0,Y 315.214,Z 514.358,A -85,B 0,C 180,E1 -15592.36,E2 -15592.36} C_VEL
LIN {X 0,Y 313.374,Z 500.639,A -85,B 0,C 180,E1 -15593.146,E2 -15593.146} C_VEL
LIN {X 0,Y 312.362,Z 493.917,A -85,B 0,C 180,E1 -15593.465,E2 -15593.465} C_VEL
LIN {X 0,Y 313.27,Z 483.658,A -85,B 0,C 180,E1 -15597.381,E2 -15597.381} C_VEL
LIN {X 0,Y 314.474,Z 473.003,A -85,B 0,C 180,E1 -15601.434,E2 -15601.434} C_VEL
LIN {X 0,Y 315.67,Z 464.073,A -85,B 0,C 180,E1 -15604.865,E2 -15604.865} C_VEL
LIN {X 0,Y 316.767,Z 457.08,A -85,B 0,C 180,E1 -15607.599,E2 -15607.599} C_VEL
LIN {X 0,Y 316.716,Z 453.541,A -85,B 0,C 180,E1 -15609.044,E2 -15609.044} C_VEL
LIN {X 0,Y 315.148,Z 445.458,A -85,B 0,C 180,E1 -15612.615,E2 -15612.615} C_VEL
LIN {X 0,Y 313.645,Z 438.253,A -85,B 0,C 180,E1 -15616.002,E2 -15616.002} C_VEL
LIN {X 0,Y 312.487,Z 432.565,A -85,B 0,C 180,E1 -15618.911,E2 -15618.911} C_VEL
LIN {X 0,Y 312.54,Z 432.554,A -85,B 0,C 180,E1 -15622.617,E2 -15622.617} C_VEL
LIN {X 0,Y 312.522,Z 432.556,A -85,B 0,C 180,E1 -15626.311,E2 -15626.311} C_VEL
LIN {X 0,Y 312.54,Z 432.555,A -85,B 0,C 180,E1 -15630.35,E2 -15630.35} C_VEL
LIN {X 0,Y 312.605,Z 432.547,A -85,B 0,C 180,E1 -15634.065,E2 -15634.065} C_VEL
LIN {X 0,Y 312.567,Z 432.55,A -85,B 0,C 180,E1 -15637.527,E2 -15637.527} C_VEL
LIN {X 0,Y 312.641,Z 432.542,A -85,B 0,C 180,E1 -15641.657,E2 -15641.657} C_VEL
LIN {X 0,Y 312.697,Z 432.537,A -85,B 0,C 180,E1 -15645.686,E2 -15645.686} C_VEL
LIN {X 0,Y 312.702,Z 432.536,A -85,B 0,C 180,E1 -15649.642,E2 -15649.642} C_VEL
LIN {X 0,Y 312.897,Z 432.512,A -85,B 0,C 180,E1 -15653.552,E2 -15653.552} C_VEL
LIN {X 0,Y 312.942,Z 432.504,A -85,B 0,C 180,E1 -15657.426,E2 -15657.426} C_VEL
LIN {X 0,Y 313.124,Z 432.48,A -85,B 0,C 180,E1 -15660,E2 -15660} C_VEL
LIN {X 0,Y 312.94,Z 432.501,A -85,B 0,C 180,E1 -15662.574,E2 -15662.574} C_VEL
LIN {X 0,Y 312.883,Z 432.507,A -85,B 0,C 180,E1 -15666.579,E2 -15666.579} C_VEL
LIN {X 0,Y 312.702,Z 432.53,A -85,B 0,C 180,E1 -15670.358,E2 -15670.358} C_VEL
LIN {X 0,Y 312.703,Z 432.521,A -85,B 0,C 180,E1 -15674.888,E2 -15674.888} C_VEL
LIN {X 0,Y 312.633,Z 432.537,A -85,B 0,C 180,E1 -15679.237,E2 -15679.237} C_VEL
LIN {X 0,Y 312.549,Z 432.55,A -85,B 0,C 180,E1 -15682.789,E2 -15682.789} C_VEL
LIN {X 0,Y 312.6,Z 432.536,A -85,B 0,C 180,E1 -15685.933,E2 -15685.933} C_VEL
LIN {X 0,Y 312.541,Z 432.549,A -85,B 0,C 180,E1 -15689.651,E2 -15689.651} C_VEL
LIN {X 0,Y 312.522,Z 432.554,A -85,B 0,C 180,E1 -15693.689,E2 -15693.689} C_VEL
LIN {X 0,Y 312.523,Z 432.556,A -85,B 0,C 180,E1 -15697.386,E2 -15697.386} C_VEL
LIN {X 0,Y 312.493,Z 432.557,A -85,B 0,C 180,E1 -15700.709,E2 -15700.709} C_VEL
LIN {X 0,Y 312.521,Z 432.552,A -85,B 0,C 180,E1 -15704.197,E2 -15704.197} C_VEL
LIN {X 0,Y 312.551,Z 432.548,A -85,B 0,C 180,E1 -15707.905,E2 -15707.905} C_VEL
LIN {X 0,Y 312.562,Z 432.547,A -85,B 0,C 180,E1 -15711.905,E2 -15711.905} C_VEL
LIN {X 0,Y 312.509,Z 432.553,A -85,B 0,C 180,E1 -15715.79,E2 -15715.79} C_VEL
LIN {X 0,Y 312.523,Z 432.556,A -85,B 0,C 180,E1 -15718.854,E2 -15718.854} C_VEL
LIN {X 0,Y 312.573,Z 432.548,A -85,B 0,C 180,E1 -15721.824,E2 -15721.824} C_VEL
LIN {X 0,Y 312.588,Z 432.548,A -85,B 0,C 180,E1 -15724.711,E2 -15724.711} C_VEL
LIN {X 0,Y 312.573,Z 432.549,A -85,B 0,C 180,E1 -15727.553,E2 -15727.553} C_VEL
LIN {X 0,Y 317.065,Z 445.048,A -85,B 0,C 180,E1 -15728.898,E2 -15728.898} C_VEL
LIN {X 0,Y 320.293,Z 455.403,A -85,B 0,C 180,E1 -15730.203,E2 -15730.203} C_VEL
LIN {X 0,Y 321.264,Z 460.156,A -85,B 0,C 180,E1 -15730.844,E2 -15730.844} C_VEL
LIN {X 0,Y 319.926,Z 470.994,A -85,B 0,C 180,E1 -15732.254,E2 -15732.254} C_VEL
LIN {X 0,Y 318.832,Z 479.754,A -85,B 0,C 180,E1 -15733.677,E2 -15733.677} C_VEL
LIN {X 0,Y 317.386,Z 489.248,A -85,B 0,C 180,E1 -15735.575,E2 -15735.575} C_VEL
LIN {X 0,Y 316.079,Z 496.82,A -85,B 0,C 180,E1 -15737.479,E2 -15737.479} C_VEL
LIN {X 0,Y 315.26,Z 502.085,A -85,B 0,C 180,E1 -15739.121,E2 -15739.121} C_VEL
LIN {X 0,Y 314.53,Z 506.93,A -85,B 0,C 180,E1 -15741.001,E2 -15741.001} C_VEL
LIN {X 0,Y 313.747,Z 510.813,A -85,B 0,C 180,E1 -15742.923,E2 -15742.923} C_VEL
LIN {X 0,Y 313.149,Z 513.68,A -85,B 0,C 180,E1 -15744.849,E2 -15744.849} C_VEL
LIN {X 0,Y 312.863,Z 515.053,A -85,B 0,C 180,E1 -15746.136,E2 -15746.136} C_VEL
LIN {X 0,Y 312.851,Z 516.583,A -85,B 0,C 180,E1 -15748.713,E2 -15748.713} C_VEL
LIN {X 0,Y 312.838,Z 516.807,A -85,B 0,C 180,E1 -15750,E2 -15750} C_VEL
LIN {X 0,Y 312.85,Z 516.623,A -85,B 0,C 180,E1 -15751.287,E2 -15751.287} C_VEL
LIN {X 0,Y 312.855,Z 515.143,A -85,B 0,C 180,E1 -15753.864,E2 -15753.864} C_VEL
LIN {X 0,Y 313.136,Z 513.812,A -85,B 0,C 180,E1 -15755.151,E2 -15755.151} C_VEL
LIN {X 0,Y 313.739,Z 510.992,A -85,B 0,C 180,E1 -15757.077,E2 -15757.077} C_VEL
LIN {X 0,Y 314.491,Z 507.174,A -85,B 0,C 180,E1 -15759,E2 -15759} C_VEL
LIN {X 0,Y 315.306,Z 501.279,A -85,B 0,C 180,E1 -15761.263,E2 -15761.263} C_VEL
LIN {X 0,Y 316.476,Z 494.867,A -85,B 0,C 180,E1 -15763.157,E2 -15763.157} C_VEL
LIN {X 0,Y 317.834,Z 486.831,A -85,B 0,C 180,E1 -15765.059,E2 -15765.059} C_VEL
LIN {X 0,Y 318.943,Z 478.612,A -85,B 0,C 180,E1 -15766.646,E2 -15766.646} C_VEL
LIN {X 0,Y 320.281,Z 468.415,A -85,B 0,C 180,E1 -15768.221,E2 -15768.221} C_VEL
LIN {X 0,Y 321.315,Z 459.716,A -85,B 0,C 180,E1 -15769.317,E2 -15769.317} C_VEL
LIN {X 0,Y 318.563,Z 449.529,A -85,B 0,C 180,E1 -15770.67,E2 -15770.67} C_VEL
LIN {X 0,Y 314.706,Z 438.303,A -85,B 0,C 180,E1 -15771.971,E2 -15771.971} C_VEL
LIN {X 0,Y 312.587,Z 432.549,A -85,B 0,C 180,E1 -15772.559,E2 -15772.559} C_VEL
LIN {X 0,Y 312.605,Z 432.544,A -85,B 0,C 180,E1 -15775.935,E2 -15775.935} C_VEL
LIN {X 0,Y 312.54,Z 432.552,A -85,B 0,C 180,E1 -15779.651,E2 -15779.651} C_VEL
LIN {X 0,Y 312.522,Z 432.554,A -85,B 0,C 180,E1 -15783.689,E2 -15783.689} C_VEL
LIN {X 0,Y 312.556,Z 432.552,A -85,B 0,C 180,E1 -15787.381,E2 -15787.381} C_VEL
LIN {X 0,Y 312.535,Z 432.554,A -85,B 0,C 180,E1 -15790.702,E2 -15790.702} C_VEL
LIN {X 0,Y 312.532,Z 432.552,A -85,B 0,C 180,E1 -15794.195,E2 -15794.195} C_VEL
LIN {X 0,Y 312.489,Z 432.557,A -85,B 0,C 180,E1 -15797.918,E2 -15797.918} C_VEL
LIN {X 0,Y 312.5,Z 432.561,A -85,B 0,C 180,E1 -15800.971,E2 -15800.971} C_VEL
LIN {X 0,Y 312.534,Z 432.552,A -85,B 0,C 180,E1 -15804.22,E2 -15804.22} C_VEL
LIN {X 0,Y 312.505,Z 432.555,A -85,B 0,C 180,E1 -15807.334,E2 -15807.334} C_VEL
LIN {X 0,Y 312.546,Z 432.551,A -85,B 0,C 180,E1 -15811.279,E2 -15811.279} C_VEL
LIN {X 0,Y 312.587,Z 432.55,A -85,B 0,C 180,E1 -15814.711,E2 -15814.711} C_VEL
LIN {X 0,Y 312.589,Z 432.543,A -85,B 0,C 180,E1 -15817.529,E2 -15817.529} C_VEL
LIN {X 0,Y 312.64,Z 432.538,A -85,B 0,C 180,E1 -15821.656,E2 -15821.656} C_VEL
LIN {X 0,Y 312.696,Z 432.531,A -85,B 0,C 180,E1 -15825.686,E2 -15825.686} C_VEL
LIN {X 0,Y 312.638,Z 432.537,A -85,B 0,C 180,E1 -15826.678,E2 -15826.678} C_VEL
LIN {X 0,Y 311.984,Z 432.623,A -85,B 0,C 180,E1 -15827.753,E2 -15827.753} C_VEL
LIN {X 0,Y 309.196,Z 432.975,A -85,B 0,C 180,E1 -15829.506,E2 -15829.506} C_VEL
LIN {X 0,Y 306.844,Z 433.267,A -85,B 0,C 180,E1 -15830.926,E2 -15830.926} C_VEL
LIN {X 0,Y 305.849,Z 433.386,A -85,B 0,C 180,E1 -15832.025,E2 -15832.025} C_VEL
LIN {X 0,Y 305.774,Z 433.393,A -85,B 0,C 180,E1 -15832.396,E2 -15832.396} C_VEL
LIN {X 0,Y 305.687,Z 433.403,A -85,B 0,C 180,E1 -15834.723,E2 -15834.723} C_VEL
LIN {X 0,Y 305.96,Z 433.373,A -85,B 0,C 180,E1 -15838.684,E2 -15838.684} C_VEL
LIN {X 0,Y 305.96,Z 433.367,A -85,B 0,C 180,E1 -15841.316,E2 -15841.316} C_VEL
LIN {X 0,Y 305.688,Z 433.405,A -85,B 0,C 180,E1 -15845.277,E2 -15845.277} C_VEL
LIN {X 0,Y 305.774,Z 433.393,A -85,B 0,C 180,E1 -15847.927,E2 -15847.927} C_VEL
LIN {X 0,Y 305.608,Z 433.417,A -85,B 0,C 180,E1 -15851.945,E2 -15851.945} C_VEL
LIN {X 0,Y 305.64,Z 433.411,A -85,B 0,C 180,E1 -15855.035,E2 -15855.035} C_VEL
LIN {X 0,Y 305.577,Z 433.419,A -85,B 0,C 180,E1 -15859.444,E2 -15859.444} C_VEL
LIN {X 0,Y 305.487,Z 433.43,A -85,B 0,C 180,E1 -15863.039,E2 -15863.039} C_VEL
LIN {X 0,Y 305.548,Z 433.427,A -85,B 0,C 180,E1 -15866.227,E2 -15866.227} C_VEL
LIN {X 0,Y 305.489,Z 433.43,A -85,B 0,C 180,E1 -15869.047,E2 -15869.047} C_VEL
LIN {X 0,Y 305.444,Z 433.439,A -85,B 0,C 180,E1 -15871.952,E2 -15871.952} C_VEL
LIN {X 0,Y 305.464,Z 433.434,A -85,B 0,C 180,E1 -15875.113,E2 -15875.113} C_VEL
LIN {X 0,Y 305.468,Z 433.435,A -85,B 0,C 180,E1 -15878.533,E2 -15878.533} C_VEL
LIN {X 0,Y 305.459,Z 433.536,A -85,B 0,C 180,E1 -15880.601,E2 -15880.601} C_VEL
LIN {X 0,Y 307.168,Z 441.832,A -85,B 0,C 180,E1 -15884.824,E2 -15884.824} C_VEL
LIN {X 0,Y 308.43,Z 448.022,A -85,B 0,C 180,E1 -15887.779,E2 -15887.779} C_VEL
LIN {X 0,Y 309.764,Z 455.131,A -85,B 0,C 180,E1 -15890.979,E2 -15890.979} C_VEL
LIN {X 0,Y 309.611,Z 459.052,A -85,B 0,C 180,E1 -15892.606,E2 -15892.606} C_VEL
LIN {X 0,Y 308.081,Z 469.58,A -85,B 0,C 180,E1 -15896.805,E2 -15896.805} C_VEL
LIN {X 0,Y 306.591,Z 480.839,A -85,B 0,C 180,E1 -15901.224,E2 -15901.224} C_VEL
LIN {X 0,Y 305.67,Z 490.027,A -85,B 0,C 180,E1 -15904.827,E2 -15904.827} C_VEL
LIN {X 0,Y 305.411,Z 493.018,A -85,B 0,C 180,E1 -15905.976,E2 -15905.976} C_VEL
LIN {X 0,Y 307.614,Z 507.47,A -85,B 0,C 180,E1 -15906.714,E2 -15906.714} C_VEL
LIN {X 0,Y 308.993,Z 520.835,A -85,B 0,C 180,E1 -15907.641,E2 -15907.641} C_VEL
LIN {X 0,Y 309.528,Z 533.508,A -85,B 0,C 180,E1 -15908.753,E2 -15908.753} C_VEL
LIN {X 0,Y 309.565,Z 544.327,A -85,B 0,C 180,E1 -15909.924,E2 -15909.924} C_VEL
LIN {X 0,Y 309.176,Z 554.661,A -85,B 0,C 180,E1 -15911.272,E2 -15911.272} C_VEL
LIN {X 0,Y 307.801,Z 564.103,A -85,B 0,C 180,E1 -15912.733,E2 -15912.733} C_VEL
LIN {X 0,Y 306.601,Z 572.457,A -85,B 0,C 180,E1 -15914.31,E2 -15914.31} C_VEL
LIN {X 0,Y 305.975,Z 577.212,A -85,B 0,C 180,E1 -15915.365,E2 -15915.365} C_VEL
LIN {X 0,Y 305.089,Z 584.856,A -85,B 0,C 180,E1 -15917.359,E2 -15917.359} C_VEL
LIN {X 0,Y 304.527,Z 591.032,A -85,B 0,C 180,E1 -15919.361,E2 -15919.361} C_VEL
LIN {X 0,Y 304.388,Z 595.965,A -85,B 0,C 180,E1 -15921.369,E2 -15921.369} C_VEL
LIN {X 0,Y 304.496,Z 599.77,A -85,B 0,C 180,E1 -15923.373,E2 -15923.373} C_VEL
LIN {X 0,Y 304.66,Z 601.748,A -85,B 0,C 180,E1 -15924.706,E2 -15924.706} C_VEL
LIN {X 0,Y 304.902,Z 603.25,A -85,B 0,C 180,E1 -15926.035,E2 -15926.035} C_VEL
LIN {X 0,Y 304.989,Z 604.309,A -85,B 0,C 180,E1 -15927.359,E2 -15927.359} C_VEL
LIN {X 0,Y 305.448,Z 605.236,A -85,B 0,C 180,E1 -15930,E2 -15930} C_VEL
LIN {X 0,Y 304.99,Z 604.3,A -85,B 0,C 180,E1 -15932.642,E2 -15932.642} C_VEL
LIN {X 0,Y 304.902,Z 603.238,A -85,B 0,C 180,E1 -15933.965,E2 -15933.965} C_VEL
LIN {X 0,Y 304.659,Z 601.73,A -85,B 0,C 180,E1 -15935.295,E2 -15935.295} C_VEL
LIN {X 0,Y 304.43,Z 599.223,A -85,B 0,C 180,E1 -15936.931,E2 -15936.931} C_VEL
LIN {X 0,Y 304.403,Z 594.423,A -85,B 0,C 180,E1 -15939.301,E2 -15939.301} C_VEL
LIN {X 0,Y 304.73,Z 588.049,A -85,B 0,C 180,E1 -15941.643,E2 -15941.643} C_VEL
LIN {X 0,Y 305.419,Z 581.153,A -85,B 0,C 180,E1 -15943.643,E2 -15943.643} C_VEL
LIN {X 0,Y 306.312,Z 573.668,A -85,B 0,C 180,E1 -15945.411,E2 -15945.411} C_VEL
LIN {X 0,Y 307.589,Z 565.838,A -85,B 0,C 180,E1 -15946.937,E2 -15946.937} C_VEL
LIN {X 0,Y 308.96,Z 555.674,A -85,B 0,C 180,E1 -15948.57,E2 -15948.57} C_VEL
LIN {X 0,Y 309.476,Z 545.552,A -85,B 0,C 180,E1 -15949.916,E2 -15949.916} C_VEL
LIN {X 0,Y 309.528,Z 533.285,A -85,B 0,C 180,E1 -15951.247,E2 -15951.247} C_VEL
LIN {X 0,Y 308.89,Z 520.059,A -85,B 0,C 180,E1 -15952.402,E2 -15952.402} C_VEL
LIN {X 0,Y 307.459,Z 506.353,A -85,B 0,C 180,E1 -15953.327,E2 -15953.327} C_VEL
LIN {X 0,Y 305.404,Z 492.874,A -85,B 0,C 180,E1 -15954.024,E2 -15954.024} C_VEL
LIN {X 0,Y 306.341,Z 482.615,A -85,B 0,C 180,E1 -15958.054,E2 -15958.054} C_VEL
LIN {X 0,Y 307.864,Z 470.764,A -85,B 0,C 180,E1 -15962.698,E2 -15962.698} C_VEL
LIN {X 0,Y 309.355,Z 460.386,A -85,B 0,C 180,E1 -15966.817,E2 -15966.817} C_VEL
LIN {X 0,Y 309.79,Z 458.02,A -85,B 0,C 180,E1 -15967.773,E2 -15967.773} C_VEL
LIN {X 0,Y 309.609,Z 454.002,A -85,B 0,C 180,E1 -15969.485,E2 -15969.485} C_VEL
LIN {X 0,Y 307.972,Z 445.852,A -85,B 0,C 180,E1 -15973.205,E2 -15973.205} C_VEL
LIN {X 0,Y 306.55,Z 438.972,A -85,B 0,C 180,E1 -15976.545,E2 -15976.545} C_VEL
LIN {X 0,Y 305.459,Z 433.44,A -85,B 0,C 180,E1 -15979.51,E2 -15979.51} C_VEL
LIN {X 0,Y 305.498,Z 433.43,A -85,B 0,C 180,E1 -15983.264,E2 -15983.264} C_VEL
LIN {X 0,Y 305.467,Z 433.434,A -85,B 0,C 180,E1 -15986.483,E2 -15986.483} C_VEL
LIN {X 0,Y 305.461,Z 433.435,A -85,B 0,C 180,E1 -15989.591,E2 -15989.591} C_VEL
LIN {X 0,Y 305.521,Z 433.429,A -85,B 0,C 180,E1 -15992.609,E2 -15992.609} C_VEL
LIN {X 0,Y 305.507,Z 433.429,A -85,B 0,C 180,E1 -15995.539,E2 -15995.539} C_VEL
LIN {X 0,Y 305.515,Z 433.431,A -85,B 0,C 180,E1 -15999.815,E2 -15999.815} C_VEL
LIN {X 0,Y 305.577,Z 433.419,A -85,B 0,C 180,E1 -16002.603,E2 -16002.603} C_VEL
LIN {X 0,Y 305.652,Z 433.412,A -85,B 0,C 180,E1 -16005.349,E2 -16005.349} C_VEL
LIN {X 0,Y 305.64,Z 433.414,A -85,B 0,C 180,E1 -16009.4,E2 -16009.4} C_VEL
LIN {X 0,Y 305.775,Z 433.397,A -85,B 0,C 180,E1 -16012.073,E2 -16012.073} C_VEL
LIN {X 0,Y 305.689,Z 433.405,A -85,B 0,C 180,E1 -16014.724,E2 -16014.724} C_VEL
LIN {X 0,Y 305.961,Z 433.371,A -85,B 0,C 180,E1 -16018.684,E2 -16018.684} C_VEL
LIN {X 0,Y 305.961,Z 433.373,A -85,B 0,C 180,E1 -16021.316,E2 -16021.316} C_VEL
LIN {X 0,Y 305.688,Z 433.407,A -85,B 0,C 180,E1 -16025.277,E2 -16025.277} C_VEL
LIN {X 0,Y 305.775,Z 433.396,A -85,B 0,C 180,E1 -16027.927,E2 -16027.927} C_VEL
LIN {X 0,Y 305.609,Z 433.411,A -85,B 0,C 180,E1 -16031.945,E2 -16031.945} C_VEL
LIN {X 0,Y 305.641,Z 433.399,A -85,B 0,C 180,E1 -16035.035,E2 -16035.035} C_VEL
LIN {X 0,Y 305.58,Z 433.417,A -85,B 0,C 180,E1 -16039.445,E2 -16039.445} C_VEL
LIN {X 0,Y 305.494,Z 433.43,A -85,B 0,C 180,E1 -16043.042,E2 -16043.042} C_VEL
LIN {X 0,Y 305.528,Z 433.415,A -85,B 0,C 180,E1 -16046.219,E2 -16046.219} C_VEL
LIN {X 0,Y 305.49,Z 433.42,A -85,B 0,C 180,E1 -16049.047,E2 -16049.047} C_VEL
LIN {X 0,Y 305.445,Z 433.434,A -85,B 0,C 180,E1 -16051.952,E2 -16051.952} C_VEL
LIN {X 0,Y 305.465,Z 433.434,A -85,B 0,C 180,E1 -16055.113,E2 -16055.113} C_VEL
LIN {X 0,Y 305.443,Z 433.436,A -85,B 0,C 180,E1 -16058.527,E2 -16058.527} C_VEL
LIN {X 0,Y 305.466,Z 433.434,A -85,B 0,C 180,E1 -16062.588,E2 -16062.588} C_VEL
LIN {X 0,Y 305.493,Z 433.429,A -85,B 0,C 180,E1 -16066.357,E2 -16066.357} C_VEL
LIN {X 0,Y 305.502,Z 433.426,A -85,B 0,C 180,E1 -16069.899,E2 -16069.899} C_VEL
LIN {X 0,Y 305.505,Z 433.426,A -85,B 0,C 180,E1 -16073.626,E2 -16073.626} C_VEL
LIN {X 0,Y 305.467,Z 433.431,A -85,B 0,C 180,E1 -16076.483,E2 -16076.483} C_VEL
LIN {X 0,Y 305.461,Z 433.433,A -85,B 0,C 180,E1 -16079.59,E2 -16079.59} C_VEL
LIN {X 0,Y 305.521,Z 433.43,A -85,B 0,C 180,E1 -16082.608,E2 -16082.608} C_VEL
LIN {X 0,Y 305.511,Z 433.428,A -85,B 0,C 180,E1 -16085.539,E2 -16085.539} C_VEL
LIN {X 0,Y 305.494,Z 433.435,A -85,B 0,C 180,E1 -16086.977,E2 -16086.977} C_VEL
LIN {X 0,Y 310.443,Z 446.979,A -85,B 0,C 180,E1 -16088.507,E2 -16088.507} C_VEL
LIN {X 0,Y 313.481,Z 456.716,A -85,B 0,C 180,E1 -16089.784,E2 -16089.784} C_VEL
LIN {X 0,Y 314.588,Z 461.173,A -85,B 0,C 180,E1 -16090.421,E2 -16090.421} C_VEL
LIN {X 0,Y 313.241,Z 472.003,A -85,B 0,C 180,E1 -16091.862,E2 -16091.862} C_VEL
LIN {X 0,Y 312.096,Z 480.762,A -85,B 0,C 180,E1 -16093.315,E2 -16093.315} C_VEL
LIN {X 0,Y 310.586,Z 490.255,A -85,B 0,C 180,E1 -16095.252,E2 -16095.252} C_VEL
LIN {X 0,Y 309.222,Z 497.827,A -85,B 0,C 180,E1 -16097.197,E2 -16097.197} C_VEL
LIN {X 0,Y 308.361,Z 503.091,A -85,B 0,C 180,E1 -16098.875,E2 -16098.875} C_VEL
LIN {X 0,Y 307.591,Z 507.936,A -85,B 0,C 180,E1 -16100.796,E2 -16100.796} C_VEL
LIN {X 0,Y 306.776,Z 511.819,A -85,B 0,C 180,E1 -16102.761,E2 -16102.761} C_VEL
LIN {X 0,Y 306.15,Z 514.686,A -85,B 0,C 180,E1 -16104.731,E2 -16104.731} C_VEL
LIN {X 0,Y 305.851,Z 516.059,A -85,B 0,C 180,E1 -16106.047,E2 -16106.047} C_VEL
LIN {X 0,Y 305.829,Z 517.588,A -85,B 0,C 180,E1 -16108.683,E2 -16108.683} C_VEL
LIN {X 0,Y 305.815,Z 517.812,A -85,B 0,C 180,E1 -16110,E2 -16110} C_VEL
LIN {X 0,Y 305.829,Z 517.627,A -85,B 0,C 180,E1 -16111.317,E2 -16111.317} C_VEL
LIN {X 0,Y 305.843,Z 516.148,A -85,B 0,C 180,E1 -16113.953,E2 -16113.953} C_VEL
LIN {X 0,Y 306.137,Z 514.816,A -85,B 0,C 180,E1 -16115.269,E2 -16115.269} C_VEL
LIN {X 0,Y 306.768,Z 511.996,A -85,B 0,C 180,E1 -16117.239,E2 -16117.239} C_VEL
LIN {X 0,Y 307.551,Z 508.178,A -85,B 0,C 180,E1 -16119.205,E2 -16119.205} C_VEL
LIN {X 0,Y 308.416,Z 502.285,A -85,B 0,C 180,E1 -16121.518,E2 -16121.518} C_VEL
LIN {X 0,Y 309.638,Z 495.87,A -85,B 0,C 180,E1 -16123.453,E2 -16123.453} C_VEL
LIN {X 0,Y 311.053,Z 487.833,A -85,B 0,C 180,E1 -16125.396,E2 -16125.396} C_VEL
LIN {X 0,Y 312.216,Z 479.614,A -85,B 0,C 180,E1 -16127.016,E2 -16127.016} C_VEL
LIN {X 0,Y 313.615,Z 469.517,A -85,B 0,C 180,E1 -16128.608,E2 -16128.608} C_VEL
LIN {X 0,Y 314.501,Z 460.565,A -85,B 0,C 180,E1 -16129.775,E2 -16129.775} C_VEL
LIN {X 0,Y 311.641,Z 450.582,A -85,B 0,C 180,E1 -16131.151,E2 -16131.151} C_VEL
LIN {X 0,Y 307.948,Z 439.835,A -85,B 0,C 180,E1 -16132.439,E2 -16132.439} C_VEL
LIN {X 0,Y 305.527,Z 433.56,A -85,B 0,C 180,E1 -16133.111,E2 -16133.111} C_VEL
LIN {X 0,Y 305.534,Z 433.424,A -85,B 0,C 180,E1 -16136.221,E2 -16136.221} C_VEL
LIN {X 0,Y 305.49,Z 433.426,A -85,B 0,C 180,E1 -16139.047,E2 -16139.047} C_VEL
LIN {X 0,Y 305.444,Z 433.433,A -85,B 0,C 180,E1 -16141.952,E2 -16141.952} C_VEL
LIN {X 0,Y 305.465,Z 433.435,A -85,B 0,C 180,E1 -16145.113,E2 -16145.113} C_VEL
LIN {X 0,Y 305.497,Z 433.43,A -85,B 0,C 180,E1 -16148.54,E2 -16148.54} C_VEL
LIN {X 0,Y 305.51,Z 433.429,A -85,B 0,C 180,E1 -16152.597,E2 -16152.597} C_VEL
LIN {X 0,Y 305.472,Z 433.432,A -85,B 0,C 180,E1 -16156.353,E2 -16156.353} C_VEL
LIN {X 0,Y 305.46,Z 433.433,A -85,B 0,C 180,E1 -16159.892,E2 -16159.892} C_VEL
LIN {X 0,Y 305.482,Z 433.43,A -85,B 0,C 180,E1 -16163.632,E2 -16163.632} C_VEL
LIN {X 0,Y 305.467,Z 433.435,A -85,B 0,C 180,E1 -16166.483,E2 -16166.483} C_VEL
LIN {X 0,Y 305.46,Z 433.434,A -85,B 0,C 180,E1 -16169.59,E2 -16169.59} C_VEL
LIN {X 0,Y 305.516,Z 433.428,A -85,B 0,C 180,E1 -16172.608,E2 -16172.608} C_VEL
LIN {X 0,Y 305.51,Z 433.427,A -85,B 0,C 180,E1 -16175.539,E2 -16175.539} C_VEL
LIN {X 0,Y 305.522,Z 433.425,A -85,B 0,C 180,E1 -16179.815,E2 -16179.815} C_VEL
LIN {X 0,Y 305.577,Z 433.421,A -85,B 0,C 180,E1 -16182.603,E2 -16182.603} C_VEL
LIN {X 0,Y 305.651,Z 433.41,A -85,B 0,C 180,E1 -16185.349,E2 -16185.349} C_VEL
LIN {X 0,Y 305.639,Z 433.41,A -85,B 0,C 180,E1 -16189.4,E2 -16189.4} C_VEL
LIN {X 0,Y 305.774,Z 433.393,A -85,B 0,C 180,E1 -16192.396,E2 -16192.396} C_VEL
LIN {X 0,Y 305.123,Z 433.473,A -85,B 0,C 180,E1 -16193.494,E2 -16193.494} C_VEL
LIN {X 0,Y 302.282,Z 433.825,A -85,B 0,C 180,E1 -16195.282,E2 -16195.282} C_VEL
LIN {X 0,Y 299.902,Z 434.128,A -85,B 0,C 180,E1 -16196.733,E2 -16196.733} C_VEL
LIN {X 0,Y 298.933,Z 434.246,A -85,B 0,C 180,E1 -16197.856,E2 -16197.856} C_VEL
LIN {X 0,Y 298.882,Z 434.252,A -85,B 0,C 180,E1 -16198.236,E2 -16198.236} C_VEL
LIN {X 0,Y 299.028,Z 434.236,A -85,B 0,C 180,E1 -16200,E2 -16200} C_VEL
LIN {X 0,Y 298.84,Z 434.259,A -85,B 0,C 180,E1 -16202.696,E2 -16202.696} C_VEL
LIN {X 0,Y 298.779,Z 434.264,A -85,B 0,C 180,E1 -16206.754,E2 -16206.754} C_VEL
LIN {X 0,Y 298.633,Z 434.283,A -85,B 0,C 180,E1 -16209.482,E2 -16209.482} C_VEL
LIN {X 0,Y 298.555,Z 434.292,A -85,B 0,C 180,E1 -16213.615,E2 -16213.615} C_VEL
LIN {X 0,Y 298.551,Z 434.295,A -85,B 0,C 180,E1 -16216.409,E2 -16216.409} C_VEL
LIN {X 0,Y 298.512,Z 434.301,A -85,B 0,C 180,E1 -16219.654,E2 -16219.654} C_VEL
LIN {X 0,Y 298.43,Z 434.311,A -85,B 0,C 180,E1 -16223.6,E2 -16223.6} C_VEL
LIN {X 0,Y 298.49,Z 434.303,A -85,B 0,C 180,E1 -16226.574,E2 -16226.574} C_VEL
LIN {X 0,Y 298.418,Z 434.313,A -85,B 0,C 180,E1 -16229.641,E2 -16229.641} C_VEL
LIN {X 0,Y 298.397,Z 434.315,A -85,B 0,C 180,E1 -16232.8,E2 -16232.8} C_VEL
LIN {X 0,Y 298.466,Z 434.307,A -85,B 0,C 180,E1 -16236.812,E2 -16236.812} C_VEL
LIN {X 0,Y 298.432,Z 434.414,A -85,B 0,C 180,E1 -16240.031,E2 -16240.031} C_VEL
LIN {X 0,Y 299.906,Z 441.721,A -85,B 0,C 180,E1 -16243.892,E2 -16243.892} C_VEL
LIN {X 0,Y 301.37,Z 448.933,A -85,B 0,C 180,E1 -16247.446,E2 -16247.446} C_VEL
LIN {X 0,Y 302.718,Z 455.822,A -85,B 0,C 180,E1 -16250.646,E2 -16250.646} C_VEL
LIN {X 0,Y 302.777,Z 459.192,A -85,B 0,C 180,E1 -16252.111,E2 -16252.111} C_VEL
LIN {X 0,Y 301.304,Z 468.567,A -85,B 0,C 180,E1 -16255.958,E2 -16255.958} C_VEL
LIN {X 0,Y 299.713,Z 479.808,A -85,B 0,C 180,E1 -16260.5,E2 -16260.5} C_VEL
LIN {X 0,Y 298.719,Z 488.973,A -85,B 0,C 180,E1 -16264.199,E2 -16264.199} C_VEL
LIN {X 0,Y 298.455,Z 491.788,A -85,B 0,C 180,E1 -16265.34,E2 -16265.34} C_VEL
LIN {X 0,Y 300.877,Z 507.748,A -85,B 0,C 180,E1 -16266.23,E2 -16266.23} C_VEL
LIN {X 0,Y 302.186,Z 520.565,A -85,B 0,C 180,E1 -16267.17,E2 -16267.17} C_VEL
LIN {X 0,Y 302.703,Z 534.061,A -85,B 0,C 180,E1 -16268.407,E2 -16268.407} C_VEL
LIN {X 0,Y 302.583,Z 546.033,A -85,B 0,C 180,E1 -16269.788,E2 -16269.788} C_VEL
LIN {X 0,Y 302.241,Z 554.794,A -85,B 0,C 180,E1 -16271.002,E2 -16271.002} C_VEL
LIN {X 0,Y 300.716,Z 564.917,A -85,B 0,C 180,E1 -16272.664,E2 -16272.664} C_VEL
LIN {X 0,Y 299.255,Z 573.72,A -85,B 0,C 180,E1 -16274.443,E2 -16274.443} C_VEL
LIN {X 0,Y 298.292,Z 581.468,A -85,B 0,C 180,E1 -16276.373,E2 -16276.373} C_VEL
LIN {X 0,Y 297.618,Z 588.115,A -85,B 0,C 180,E1 -16278.421,E2 -16278.421} C_VEL
LIN {X 0,Y 297.322,Z 593.439,A -85,B 0,C 180,E1 -16280.476,E2 -16280.476} C_VEL
LIN {X 0,Y 297.384,Z 598.417,A -85,B 0,C 180,E1 -16283.014,E2 -16283.014} C_VEL
LIN {X 0,Y 297.573,Z 600.731,A -85,B 0,C 180,E1 -16284.579,E2 -16284.579} C_VEL
LIN {X 0,Y 297.849,Z 602.239,A -85,B 0,C 180,E1 -16285.941,E2 -16285.941} C_VEL
LIN {X 0,Y 297.941,Z 603.3,A -85,B 0,C 180,E1 -16287.296,E2 -16287.296} C_VEL
LIN {X 0,Y 298.417,Z 604.23,A -85,B 0,C 180,E1 -16290,E2 -16290} C_VEL
LIN {X 0,Y 297.942,Z 603.29,A -85,B 0,C 180,E1 -16292.704,E2 -16292.704} C_VEL
LIN {X 0,Y 297.849,Z 602.226,A -85,B 0,C 180,E1 -16294.059,E2 -16294.059} C_VEL
LIN {X 0,Y 297.569,Z 600.711,A -85,B 0,C 180,E1 -16295.421,E2 -16295.421} C_VEL
LIN {X 0,Y 297.342,Z 597.585,A -85,B 0,C 180,E1 -16297.469,E2 -16297.469} C_VEL
LIN {X 0,Y 297.323,Z 593.396,A -85,B 0,C 180,E1 -16299.524,E2 -16299.524} C_VEL
LIN {X 0,Y 297.728,Z 587.025,A -85,B 0,C 180,E1 -16301.92,E2 -16301.92} C_VEL
LIN {X 0,Y 298.479,Z 580.129,A -85,B 0,C 180,E1 -16303.966,E2 -16303.966} C_VEL
LIN {X 0,Y 299.299,Z 573.493,A -85,B 0,C 180,E1 -16305.587,E2 -16305.587} C_VEL
LIN {X 0,Y 300.715,Z 564.806,A -85,B 0,C 180,E1 -16307.337,E2 -16307.337} C_VEL
LIN {X 0,Y 302.197,Z 554.649,A -85,B 0,C 180,E1 -16309.001,E2 -16309.001} C_VEL
LIN {X 0,Y 302.666,Z 543.252,A -85,B 0,C 180,E1 -16310.536,E2 -16310.536} C_VEL
LIN {X 0,Y 302.659,Z 531.65,A -85,B 0,C 180,E1 -16311.81,E2 -16311.81} C_VEL
LIN {X 0,Y 302.044,Z 519.188,A -85,B 0,C 180,E1 -16312.923,E2 -16312.923} C_VEL
LIN {X 0,Y 300.595,Z 505.684,A -85,B 0,C 180,E1 -16313.872,E2 -16313.872} C_VEL
LIN {X 0,Y 298.456,Z 491.842,A -85,B 0,C 180,E1 -16314.614,E2 -16314.614} C_VEL
LIN {X 0,Y 299.468,Z 481.585,A -85,B 0,C 180,E1 -16318.757,E2 -16318.757} C_VEL
LIN {X 0,Y 301.065,Z 470.263,A -85,B 0,C 180,E1 -16323.323,E2 -16323.323} C_VEL
LIN {X 0,Y 302.791,Z 459.106,A -85,B 0,C 180,E1 -16327.892,E2 -16327.892} C_VEL
LIN {X 0,Y 302.718,Z 455.749,A -85,B 0,C 180,E1 -16329.354,E2 -16329.354} C_VEL
LIN {X 0,Y 301.118,Z 447.756,A -85,B 0,C 180,E1 -16333.086,E2 -16333.086} C_VEL
LIN {X 0,Y 299.655,Z 440.613,A -85,B 0,C 180,E1 -16336.641,E2 -16336.641} C_VEL
LIN {X 0,Y 298.419,Z 434.317,A -85,B 0,C 180,E1 -16340.077,E2 -16340.077} C_VEL
LIN {X 0,Y 298.434,Z 434.314,A -85,B 0,C 180,E1 -16343.932,E2 -16343.932} C_VEL
LIN {X 0,Y 298.397,Z 434.318,A -85,B 0,C 180,E1 -16347.984,E2 -16347.984} C_VEL
LIN {X 0,Y 298.461,Z 434.31,A -85,B 0,C 180,E1 -16351.904,E2 -16351.904} C_VEL
LIN {X 0,Y 298.486,Z 434.301,A -85,B 0,C 180,E1 -16354.924,E2 -16354.924} C_VEL
LIN {X 0,Y 298.443,Z 434.308,A -85,B 0,C 180,E1 -16359.315,E2 -16359.315} C_VEL
LIN {X 0,Y 298.541,Z 434.298,A -85,B 0,C 180,E1 -16362.18,E2 -16362.18} C_VEL
LIN {X 0,Y 298.597,Z 434.29,A -85,B 0,C 180,E1 -16364.995,E2 -16364.995} C_VEL
LIN {X 0,Y 298.596,Z 434.29,A -85,B 0,C 180,E1 -16369.147,E2 -16369.147} C_VEL
LIN {X 0,Y 298.721,Z 434.278,A -85,B 0,C 180,E1 -16371.885,E2 -16371.885} C_VEL
LIN {X 0,Y 298.659,Z 434.281,A -85,B 0,C 180,E1 -16374.599,E2 -16374.599} C_VEL
LIN {X 0,Y 298.928,Z 434.247,A -85,B 0,C 180,E1 -16378.653,E2 -16378.653} C_VEL
LIN {X 0,Y 298.927,Z 434.249,A -85,B 0,C 180,E1 -16381.347,E2 -16381.347} C_VEL
LIN {X 0,Y 298.78,Z 434.265,A -85,B 0,C 180,E1 -16386.754,E2 -16386.754} C_VEL
LIN {X 0,Y 298.634,Z 434.288,A -85,B 0,C 180,E1 -16389.482,E2 -16389.482} C_VEL
LIN {X 0,Y 298.557,Z 434.282,A -85,B 0,C 180,E1 -16393.615,E2 -16393.615} C_VEL
LIN {X 0,Y 298.552,Z 434.277,A -85,B 0,C 180,E1 -16396.409,E2 -16396.409} C_VEL
LIN {X 0,Y 298.515,Z 434.299,A -85,B 0,C 180,E1 -16399.655,E2 -16399.655} C_VEL
LIN {X 0,Y 298.461,Z 434.304,A -85,B 0,C 180,E1 -16403.598,E2 -16403.598} C_VEL
LIN {X 0,Y 298.488,Z 434.291,A -85,B 0,C 180,E1 -16406.575,E2 -16406.575} C_VEL
LIN {X 0,Y 298.419,Z 434.307,A -85,B 0,C 180,E1 -16409.641,E2 -16409.641} C_VEL
LIN {X 0,Y 298.397,Z 434.314,A -85,B 0,C 180,E1 -16412.8,E2 -16412.8} C_VEL
LIN {X 0,Y 298.447,Z 434.307,A -85,B 0,C 180,E1 -16416.807,E2 -16416.807} C_VEL
LIN {X 0,Y 298.391,Z 434.317,A -85,B 0,C 180,E1 -16421.088,E2 -16421.088} C_VEL
LIN {X 0,Y 298.419,Z 434.313,A -85,B 0,C 180,E1 -16424.953,E2 -16424.953} C_VEL
LIN {X 0,Y 298.457,Z 434.307,A -85,B 0,C 180,E1 -16428.75,E2 -16428.75} C_VEL
LIN {X 0,Y 298.451,Z 434.305,A -85,B 0,C 180,E1 -16432.247,E2 -16432.247} C_VEL
LIN {X 0,Y 298.411,Z 434.309,A -85,B 0,C 180,E1 -16435.581,E2 -16435.581} C_VEL
LIN {X 0,Y 298.394,Z 434.315,A -85,B 0,C 180,E1 -16438.791,E2 -16438.791} C_VEL
LIN {X 0,Y 298.462,Z 434.306,A -85,B 0,C 180,E1 -16441.904,E2 -16441.904} C_VEL
LIN {X 0,Y 298.488,Z 434.303,A -85,B 0,C 180,E1 -16444.924,E2 -16444.924} C_VEL
LIN {X 0,Y 298.47,Z 434.307,A -85,B 0,C 180,E1 -16446.403,E2 -16446.403} C_VEL
LIN {X 0,Y 300.21,Z 439.158,A -85,B 0,C 180,E1 -16446.917,E2 -16446.917} C_VEL
LIN {X 0,Y 303.933,Z 449.258,A -85,B 0,C 180,E1 -16448.143,E2 -16448.143} C_VEL
LIN {X 0,Y 307.001,Z 459.194,A -85,B 0,C 180,E1 -16449.519,E2 -16449.519} C_VEL
LIN {X 0,Y 307.772,Z 462.214,A -85,B 0,C 180,E1 -16449.969,E2 -16449.969} C_VEL
LIN {X 0,Y 307.285,Z 467.985,A -85,B 0,C 180,E1 -16450.729,E2 -16450.729} C_VEL
LIN {X 0,Y 305.887,Z 478.079,A -85,B 0,C 180,E1 -16452.276,E2 -16452.276} C_VEL
LIN {X 0,Y 304.585,Z 486.776,A -85,B 0,C 180,E1 -16453.925,E2 -16453.925} C_VEL
LIN {X 0,Y 303.025,Z 495.274,A -85,B 0,C 180,E1 -16455.905,E2 -16455.905} C_VEL
LIN {X 0,Y 301.664,Z 502.599,A -85,B 0,C 180,E1 -16458.097,E2 -16458.097} C_VEL
LIN {X 0,Y 300.908,Z 507.393,A -85,B 0,C 180,E1 -16459.911,E2 -16459.911} C_VEL
LIN {X 0,Y 299.983,Z 511.636,A -85,B 0,C 180,E1 -16461.919,E2 -16461.919} C_VEL
LIN {X 0,Y 299.535,Z 513.871,A -85,B 0,C 180,E1 -16463.263,E2 -16463.263} C_VEL
LIN {X 0,Y 299.152,Z 515.692,A -85,B 0,C 180,E1 -16464.608,E2 -16464.608} C_VEL
LIN {X 0,Y 298.841,Z 517.064,A -85,B 0,C 180,E1 -16465.954,E2 -16465.954} C_VEL
LIN {X 0,Y 298.807,Z 518.593,A -85,B 0,C 180,E1 -16468.652,E2 -16468.652} C_VEL
LIN {X 0,Y 298.791,Z 518.816,A -85,B 0,C 180,E1 -16470,E2 -16470} C_VEL
LIN {X 0,Y 298.806,Z 518.631,A -85,B 0,C 180,E1 -16471.348,E2 -16471.348} C_VEL
LIN {X 0,Y 298.832,Z 517.153,A -85,B 0,C 180,E1 -16474.046,E2 -16474.046} C_VEL
LIN {X 0,Y 299.138,Z 515.821,A -85,B 0,C 180,E1 -16475.392,E2 -16475.392} C_VEL
LIN {X 0,Y 299.798,Z 513,A -85,B 0,C 180,E1 -16477.408,E2 -16477.408} C_VEL
LIN {X 0,Y 300.616,Z 509.182,A -85,B 0,C 180,E1 -16479.419,E2 -16479.419} C_VEL
LIN {X 0,Y 301.542,Z 503.261,A -85,B 0,C 180,E1 -16481.793,E2 -16481.793} C_VEL
LIN {X 0,Y 303.019,Z 495.673,A -85,B 0,C 180,E1 -16484.095,E2 -16484.095} C_VEL
LIN {X 0,Y 304.52,Z 487.308,A -85,B 0,C 180,E1 -16486.078,E2 -16486.078} C_VEL
LIN {X 0,Y 305.763,Z 478.724,A -85,B 0,C 180,E1 -16487.731,E2 -16487.731} C_VEL
LIN {X 0,Y 307.2,Z 468.542,A -85,B 0,C 180,E1 -16489.309,E2 -16489.309} C_VEL
LIN {X 0,Y 307.901,Z 463.085,A -85,B 0,C 180,E1 -16490.022,E2 -16490.022} C_VEL
LIN {X 0,Y 305.552,Z 454.204,A -85,B 0,C 180,E1 -16491.31,E2 -16491.31} C_VEL
LIN {X 0,Y 301.846,Z 443.109,A -85,B 0,C 180,E1 -16492.727,E2 -16492.727} C_VEL
LIN {X 0,Y 298.528,Z 434.67,A -85,B 0,C 180,E1 -16493.684,E2 -16493.684} C_VEL
LIN {X 0,Y 298.482,Z 434.305,A -85,B 0,C 180,E1 -16493.78,E2 -16493.78} C_VEL
LIN {X 0,Y 298.488,Z 434.303,A -85,B 0,C 180,E1 -16496.574,E2 -16496.574} C_VEL
LIN {X 0,Y 298.418,Z 434.311,A -85,B 0,C 180,E1 -16499.641,E2 -16499.641} C_VEL
LIN {X 0,Y 298.397,Z 434.312,A -85,B 0,C 180,E1 -16502.8,E2 -16502.8} C_VEL
LIN {X 0,Y 298.473,Z 434.306,A -85,B 0,C 180,E1 -16506.814,E2 -16506.814} C_VEL
LIN {X 0,Y 298.457,Z 434.311,A -85,B 0,C 180,E1 -16511.103,E2 -16511.103} C_VEL
LIN {X 0,Y 298.461,Z 434.309,A -85,B 0,C 180,E1 -16513.116,E2 -16513.116} C_VEL
LIN {X 0,Y 298.433,Z 434.314,A -85,B 0,C 180,E1 -16516.926,E2 -16516.926} C_VEL
LIN {X 0,Y 298.4,Z 434.317,A -85,B 0,C 180,E1 -16521.007,E2 -16521.007} C_VEL
LIN {X 0,Y 298.419,Z 434.309,A -85,B 0,C 180,E1 -16523.93,E2 -16523.93} C_VEL
LIN {X 0,Y 298.395,Z 434.311,A -85,B 0,C 180,E1 -16527.984,E2 -16527.984} C_VEL
LIN {X 0,Y 298.459,Z 434.304,A -85,B 0,C 180,E1 -16531.904,E2 -16531.904} C_VEL
LIN {X 0,Y 298.485,Z 434.305,A -85,B 0,C 180,E1 -16534.924,E2 -16534.924} C_VEL
LIN {X 0,Y 298.452,Z 434.307,A -85,B 0,C 180,E1 -16539.315,E2 -16539.315} C_VEL
LIN {X 0,Y 298.54,Z 434.296,A -85,B 0,C 180,E1 -16542.179,E2 -16542.179} C_VEL
LIN {X 0,Y 298.596,Z 434.29,A -85,B 0,C 180,E1 -16544.995,E2 -16544.995} C_VEL
LIN {X 0,Y 298.595,Z 434.288,A -85,B 0,C 180,E1 -16549.147,E2 -16549.147} C_VEL
LIN {X 0,Y 298.723,Z 434.269,A -85,B 0,C 180,E1 -16552.404,E2 -16552.404} C_VEL
LIN {X 0,Y 298.84,Z 434.257,A -85,B 0,C 180,E1 -16557.304,E2 -16557.304} C_VEL
LIN {X 0,Y 298.882,Z 434.252,A -85,B 0,C 180,E1 -16558.236,E2 -16558.236} C_VEL
LIN {X 0,Y 298.609,Z 434.29,A -85,B 0,C 180,E1 -16558.989,E2 -16558.989} C_VEL
LIN {X 0,Y 297.249,Z 434.465,A -85,B 0,C 180,E1 -16560.098,E2 -16560.098} C_VEL
LIN {X 0,Y 292.745,Z 435.027,A -85,B 0,C 180,E1 -16562.673,E2 -16562.673} C_VEL
LIN {X 0,Y 291.644,Z 435.158,A -85,B 0,C 180,E1 -16563.826,E2 -16563.826} C_VEL
LIN {X 0,Y 291.556,Z 435.166,A -85,B 0,C 180,E1 -16564.218,E2 -16564.218} C_VEL
LIN {X 0,Y 291.726,Z 435.141,A -85,B 0,C 180,E1 -16566.918,E2 -16566.918} C_VEL
LIN {X 0,Y 291.574,Z 435.163,A -85,B 0,C 180,E1 -16569.714,E2 -16569.714} C_VEL
LIN {X 0,Y 291.525,Z 435.17,A -85,B 0,C 180,E1 -16573.95,E2 -16573.95} C_VEL
LIN {X 0,Y 291.489,Z 435.172,A -85,B 0,C 180,E1 -16576.818,E2 -16576.818} C_VEL
LIN {X 0,Y 291.452,Z 435.182,A -85,B 0,C 180,E1 -16579.875,E2 -16579.875} C_VEL
LIN {X 0,Y 291.385,Z 435.191,A -85,B 0,C 180,E1 -16584.207,E2 -16584.207} C_VEL
LIN {X 0,Y 291.422,Z 435.183,A -85,B 0,C 180,E1 -16587.272,E2 -16587.272} C_VEL
LIN {X 0,Y 291.336,Z 435.196,A -85,B 0,C 180,E1 -16590.437,E2 -16590.437} C_VEL
LIN {X 0,Y 291.346,Z 435.196,A -85,B 0,C 180,E1 -16593.698,E2 -16593.698} C_VEL
LIN {X 0,Y 291.395,Z 435.188,A -85,B 0,C 180,E1 -16597.259,E2 -16597.259} C_VEL
LIN {X 0,Y 291.398,Z 435.392,A -85,B 0,C 180,E1 -16599.486,E2 -16599.486} C_VEL
LIN {X 0,Y 292.759,Z 442.044,A -85,B 0,C 180,E1 -16603.138,E2 -16603.138} C_VEL
LIN {X 0,Y 294.234,Z 449.224,A -85,B 0,C 180,E1 -16606.799,E2 -16606.799} C_VEL
LIN {X 0,Y 295.528,Z 455.97,A -85,B 0,C 180,E1 -16610.052,E2 -16610.052} C_VEL
LIN {X 0,Y 295.851,Z 459.425,A -85,B 0,C 180,E1 -16611.621,E2 -16611.621} C_VEL
LIN {X 0,Y 294.744,Z 466.41,A -85,B 0,C 180,E1 -16614.589,E2 -16614.589} C_VEL
LIN {X 0,Y 293.385,Z 475.05,A -85,B 0,C 180,E1 -16618.197,E2 -16618.197} C_VEL
LIN {X 0,Y 292.013,Z 486.106,A -85,B 0,C 180,E1 -16622.788,E2 -16622.788} C_VEL
LIN {X 0,Y 291.5,Z 490.777,A -85,B 0,C 180,E1 -16624.735,E2 -16624.735} C_VEL
LIN {X 0,Y 293.82,Z 505.506,A -85,B 0,C 180,E1 -16625.56,E2 -16625.56} C_VEL
LIN {X 0,Y 295.22,Z 518.477,A -85,B 0,C 180,E1 -16626.518,E2 -16626.518} C_VEL
LIN {X 0,Y 295.787,Z 530.828,A -85,B 0,C 180,E1 -16627.656,E2 -16627.656} C_VEL
LIN {X 0,Y 295.819,Z 542.557,A -85,B 0,C 180,E1 -16628.987,E2 -16628.987} C_VEL
LIN {X 0,Y 295.408,Z 553.762,A -85,B 0,C 180,E1 -16630.545,E2 -16630.545} C_VEL
LIN {X 0,Y 293.847,Z 563.889,A -85,B 0,C 180,E1 -16632.245,E2 -16632.245} C_VEL
LIN {X 0,Y 292.362,Z 572.976,A -85,B 0,C 180,E1 -16634.13,E2 -16634.13} C_VEL
LIN {X 0,Y 291.341,Z 580.446,A -85,B 0,C 180,E1 -16636.041,E2 -16636.041} C_VEL
LIN {X 0,Y 290.615,Z 587.094,A -85,B 0,C 180,E1 -16638.138,E2 -16638.138} C_VEL
LIN {X 0,Y 290.263,Z 592.416,A -85,B 0,C 180,E1 -16640.242,E2 -16640.242} C_VEL
LIN {X 0,Y 290.276,Z 596.596,A -85,B 0,C 180,E1 -16642.348,E2 -16642.348} C_VEL
LIN {X 0,Y 290.486,Z 599.713,A -85,B 0,C 180,E1 -16644.447,E2 -16644.447} C_VEL
LIN {X 0,Y 290.775,Z 601.225,A -85,B 0,C 180,E1 -16645.842,E2 -16645.842} C_VEL
LIN {X 0,Y 290.892,Z 602.291,A -85,B 0,C 180,E1 -16647.23,E2 -16647.23} C_VEL
LIN {X 0,Y 291.385,Z 603.224,A -85,B 0,C 180,E1 -16650,E2 -16650} C_VEL
LIN {X 0,Y 290.892,Z 602.281,A -85,B 0,C 180,E1 -16652.77,E2 -16652.77} C_VEL
LIN {X 0,Y 290.774,Z 601.211,A -85,B 0,C 180,E1 -16654.158,E2 -16654.158} C_VEL
LIN {X 0,Y 290.478,Z 599.691,A -85,B 0,C 180,E1 -16655.554,E2 -16655.554} C_VEL
LIN {X 0,Y 290.277,Z 596.565,A -85,B 0,C 180,E1 -16657.652,E2 -16657.652} C_VEL
LIN {X 0,Y 290.264,Z 592.371,A -85,B 0,C 180,E1 -16659.758,E2 -16659.758} C_VEL
LIN {X 0,Y 290.744,Z 586.002,A -85,B 0,C 180,E1 -16662.211,E2 -16662.211} C_VEL
LIN {X 0,Y 291.552,Z 579.105,A -85,B 0,C 180,E1 -16664.305,E2 -16664.305} C_VEL
LIN {X 0,Y 292.21,Z 573.593,A -85,B 0,C 180,E1 -16665.709,E2 -16665.709} C_VEL
LIN {X 0,Y 293.611,Z 565.599,A -85,B 0,C 180,E1 -16667.41,E2 -16667.41} C_VEL
LIN {X 0,Y 295.065,Z 555.794,A -85,B 0,C 180,E1 -16669.118,E2 -16669.118} C_VEL
LIN {X 0,Y 295.658,Z 546.146,A -85,B 0,C 180,E1 -16670.525,E2 -16670.525} C_VEL
LIN {X 0,Y 295.855,Z 534.219,A -85,B 0,C 180,E1 -16671.966,E2 -16671.966} C_VEL
LIN {X 0,Y 295.401,Z 521.428,A -85,B 0,C 180,E1 -16673.206,E2 -16673.206} C_VEL
LIN {X 0,Y 294.056,Z 507.377,A -85,B 0,C 180,E1 -16674.288,E2 -16674.288} C_VEL
LIN {X 0,Y 291.969,Z 493.772,A -85,B 0,C 180,E1 -16675.089,E2 -16675.089} C_VEL
LIN {X 0,Y 291.504,Z 490.77,A -85,B 0,C 180,E1 -16675.241,E2 -16675.241} C_VEL
LIN {X 0,Y 292.871,Z 478.756,A -85,B 0,C 180,E1 -16680.244,E2 -16680.244} C_VEL
LIN {X 0,Y 294.282,Z 469.361,A -85,B 0,C 180,E1 -16684.141,E2 -16684.141} C_VEL
LIN {X 0,Y 295.85,Z 459.33,A -85,B 0,C 180,E1 -16688.379,E2 -16688.379} C_VEL
LIN {X 0,Y 295.524,Z 455.894,A -85,B 0,C 180,E1 -16689.949,E2 -16689.949} C_VEL
LIN {X 0,Y 293.801,Z 447.258,A -85,B 0,C 180,E1 -16694.141,E2 -16694.141} C_VEL
LIN {X 0,Y 292.214,Z 439.46,A -85,B 0,C 180,E1 -16698.209,E2 -16698.209} C_VEL
LIN {X 0,Y 291.389,Z 435.194,A -85,B 0,C 180,E1 -16700.639,E2 -16700.639} C_VEL
LIN {X 0,Y 291.427,Z 435.184,A -85,B 0,C 180,E1 -16702.922,E2 -16702.922} C_VEL
LIN {X 0,Y 291.347,Z 435.193,A -85,B 0,C 180,E1 -16706.302,E2 -16706.302} C_VEL
LIN {X 0,Y 291.386,Z 435.192,A -85,B 0,C 180,E1 -16710.261,E2 -16710.261} C_VEL
LIN {X 0,Y 291.418,Z 435.184,A -85,B 0,C 180,E1 -16714.272,E2 -16714.272} C_VEL
LIN {X 0,Y 291.377,Z 435.189,A -85,B 0,C 180,E1 -16717.299,E2 -16717.299} C_VEL
LIN {X 0,Y 291.46,Z 435.179,A -85,B 0,C 180,E1 -16720.27,E2 -16720.27} C_VEL
LIN {X 0,Y 291.558,Z 435.167,A -85,B 0,C 180,E1 -16724.624,E2 -16724.624} C_VEL
LIN {X 0,Y 291.54,Z 435.169,A -85,B 0,C 180,E1 -16728.881,E2 -16728.881} C_VEL
LIN {X 0,Y 291.671,Z 435.156,A -85,B 0,C 180,E1 -16731.687,E2 -16731.687} C_VEL
LIN {X 0,Y 291.629,Z 435.157,A -85,B 0,C 180,E1 -16734.468,E2 -16734.468} C_VEL
LIN {X 0,Y 291.894,Z 435.124,A -85,B 0,C 180,E1 -16738.62,E2 -16738.62} C_VEL
LIN {X 0,Y 291.893,Z 435.126,A -85,B 0,C 180,E1 -16741.38,E2 -16741.38} C_VEL
LIN {X 0,Y 291.727,Z 435.144,A -85,B 0,C 180,E1 -16746.918,E2 -16746.918} C_VEL
LIN {X 0,Y 291.576,Z 435.165,A -85,B 0,C 180,E1 -16749.714,E2 -16749.714} C_VEL
LIN {X 0,Y 291.526,Z 435.154,A -85,B 0,C 180,E1 -16753.95,E2 -16753.95} C_VEL
LIN {X 0,Y 291.49,Z 435.155,A -85,B 0,C 180,E1 -16756.818,E2 -16756.818} C_VEL
LIN {X 0,Y 291.453,Z 435.176,A -85,B 0,C 180,E1 -16759.875,E2 -16759.875} C_VEL
LIN {X 0,Y 291.402,Z 435.18,A -85,B 0,C 180,E1 -16764.205,E2 -16764.205} C_VEL
LIN {X 0,Y 291.421,Z 435.167,A -85,B 0,C 180,E1 -16767.272,E2 -16767.272} C_VEL
LIN {X 0,Y 291.337,Z 435.187,A -85,B 0,C 180,E1 -16770.437,E2 -16770.437} C_VEL
LIN {X 0,Y 291.347,Z 435.191,A -85,B 0,C 180,E1 -16773.698,E2 -16773.698} C_VEL
LIN {X 0,Y 291.375,Z 435.192,A -85,B 0,C 180,E1 -16777.253,E2 -16777.253} C_VEL
LIN {X 0,Y 291.336,Z 435.192,A -85,B 0,C 180,E1 -16780.642,E2 -16780.642} C_VEL
LIN {X 0,Y 291.344,Z 435.19,A -85,B 0,C 180,E1 -16784.392,E2 -16784.392} C_VEL
LIN {X 0,Y 291.391,Z 435.185,A -85,B 0,C 180,E1 -16788.39,E2 -16788.39} C_VEL
LIN {X 0,Y 291.391,Z 435.187,A -85,B 0,C 180,E1 -16791.164,E2 -16791.164} C_VEL
LIN {X 0,Y 291.389,Z 435.186,A -85,B 0,C 180,E1 -16794.63,E2 -16794.63} C_VEL
LIN {X 0,Y 291.373,Z 435.187,A -85,B 0,C 180,E1 -16797.951,E2 -16797.951} C_VEL
LIN {X 0,Y 291.381,Z 435.191,A -85,B 0,C 180,E1 -16801.158,E2 -16801.158} C_VEL
LIN {X 0,Y 291.451,Z 435.178,A -85,B 0,C 180,E1 -16805.039,E2 -16805.039} C_VEL
LIN {X 0,Y 291.453,Z 435.384,A -85,B 0,C 180,E1 -16805.799,E2 -16805.799} C_VEL
LIN {X 0,Y 295.787,Z 446.764,A -85,B 0,C 180,E1 -16807.147,E2 -16807.147} C_VEL
LIN {X 0,Y 299.291,Z 457.233,A -85,B 0,C 180,E1 -16808.584,E2 -16808.584} C_VEL
LIN {X 0,Y 301.173,Z 464.5,A -85,B 0,C 180,E1 -16809.684,E2 -16809.684} C_VEL
LIN {X 0,Y 299.773,Z 475.067,A -85,B 0,C 180,E1 -16811.194,E2 -16811.194} C_VEL
LIN {X 0,Y 298.379,Z 484.523,A -85,B 0,C 180,E1 -16812.877,E2 -16812.877} C_VEL
LIN {X 0,Y 297.017,Z 492.27,A -85,B 0,C 180,E1 -16814.562,E2 -16814.562} C_VEL
LIN {X 0,Y 295.532,Z 499.841,A -85,B 0,C 180,E1 -16816.593,E2 -16816.593} C_VEL
LIN {X 0,Y 294.582,Z 505.105,A -85,B 0,C 180,E1 -16818.347,E2 -16818.347} C_VEL
LIN {X 0,Y 293.724,Z 509.949,A -85,B 0,C 180,E1 -16820.358,E2 -16820.358} C_VEL
LIN {X 0,Y 292.84,Z 513.831,A -85,B 0,C 180,E1 -16822.415,E2 -16822.415} C_VEL
LIN {X 0,Y 292.155,Z 516.698,A -85,B 0,C 180,E1 -16824.478,E2 -16824.478} C_VEL
LIN {X 0,Y 291.83,Z 518.07,A -85,B 0,C 180,E1 -16825.857,E2 -16825.857} C_VEL
LIN {X 0,Y 291.784,Z 519.598,A -85,B 0,C 180,E1 -16828.62,E2 -16828.62} C_VEL
LIN {X 0,Y 291.767,Z 519.821,A -85,B 0,C 180,E1 -16830,E2 -16830} C_VEL
LIN {X 0,Y 291.784,Z 519.636,A -85,B 0,C 180,E1 -16831.38,E2 -16831.38} C_VEL
LIN {X 0,Y 291.822,Z 518.157,A -85,B 0,C 180,E1 -16834.143,E2 -16834.143} C_VEL
LIN {X 0,Y 292.142,Z 516.825,A -85,B 0,C 180,E1 -16835.522,E2 -16835.522} C_VEL
LIN {X 0,Y 292.831,Z 514.004,A -85,B 0,C 180,E1 -16837.585,E2 -16837.585} C_VEL
LIN {X 0,Y 293.685,Z 510.186,A -85,B 0,C 180,E1 -16839.643,E2 -16839.643} C_VEL
LIN {X 0,Y 294.665,Z 504.268,A -85,B 0,C 180,E1 -16842.071,E2 -16842.071} C_VEL
LIN {X 0,Y 295.986,Z 497.876,A -85,B 0,C 180,E1 -16844.086,E2 -16844.086} C_VEL
LIN {X 0,Y 297.525,Z 489.839,A -85,B 0,C 180,E1 -16846.114,E2 -16846.114} C_VEL
LIN {X 0,Y 298.803,Z 481.618,A -85,B 0,C 180,E1 -16847.804,E2 -16847.804} C_VEL
LIN {X 0,Y 300.317,Z 471.742,A -85,B 0,C 180,E1 -16849.429,E2 -16849.429} C_VEL
LIN {X 0,Y 301.127,Z 464.113,A -85,B 0,C 180,E1 -16850.492,E2 -16850.492} C_VEL
LIN {X 0,Y 298.372,Z 454.328,A -85,B 0,C 180,E1 -16851.958,E2 -16851.958} C_VEL
LIN {X 0,Y 295.252,Z 445.048,A -85,B 0,C 180,E1 -16853.186,E2 -16853.186} C_VEL
LIN {X 0,Y 291.47,Z 435.431,A -85,B 0,C 180,E1 -16854.317,E2 -16854.317} C_VEL
LIN {X 0,Y 291.419,Z 435.184,A -85,B 0,C 180,E1 -16854.393,E2 -16854.393} C_VEL
LIN {X 0,Y 291.422,Z 435.181,A -85,B 0,C 180,E1 -16857.272,E2 -16857.272} C_VEL
LIN {X 0,Y 291.336,Z 435.191,A -85,B 0,C 180,E1 -16860.437,E2 -16860.437} C_VEL
